// TwinCAT 3 PLC project Perlage_Standard
// libraries:
//   Recipe Management, * (System)
//   Tc2_Drive, * (Beckhoff Automation GmbH)
//   Tc2_EtherCAT, * (Beckhoff Automation GmbH)
//   Tc2_Math, * (Beckhoff Automation GmbH)
//   Tc2_MC2, * (Beckhoff Automation GmbH)
//   Tc2_MC2_Drive, * (Beckhoff Automation GmbH)
//   Tc2_NC, * (Beckhoff Automation GmbH)
//   Tc2_SerialCom, * (Beckhoff Automation GmbH)
//   Tc2_Standard, * (Beckhoff Automation GmbH)
//   Tc2_Standard, * (Beckhoff Automation GmbH)
//   Tc2_System, * (Beckhoff Automation GmbH)
//   Tc2_System, * (Beckhoff Automation GmbH)
//   Tc2_Utilities, * (Beckhoff Automation GmbH)
//   Tc3_Module, * (Beckhoff Automation GmbH)
//   Tc3_Module, * (Beckhoff Automation GmbH)
// project tree:
//   Data types/ TAutoSampling.TcDUT, TAxisCommands.TcDUT, TAxisHomingType.TcDUT, TAxisState.TcDUT, TAxisType.TcDUT, TComIndex.TcDUT, TConfigFileData.TcDUT, TCounter.TcDUT, TDashboardCmd.TcDUT, TDataLog.TcDUT, TDynAxisParam.TcDUT, TErrors.TcDUT, TGiver.TcDUT, THolderIndex.TcDUT, TLiftPos.TcDUT, TLiftType.TcDUT, TLoaderAxis.TcDUT, TLoaderDropMode.TcDUT, TLoaderHead.TcDUT, TLoaderModulePos.TcDUT, TLoaderPlatePos.TcDUT, TLoaderSynchro.TcDUT, TLoaderTakeMode.TcDUT, TLoaderTeachedAxis.TcDUT, TLoaderTeachOffset.TcDUT, TLoaderTeachPos.TcDUT, TMachineData.TcDUT, TMachineManual.TcDUT, TMachineMode.TcDUT, TMachineModeMask.TcDUT, TMachineOptions.TcDUT, TMachineSafety.TcDUT, TManagerPartStatus.TcDUT, TManBarrel.TcDUT, TManBarrelAxisPosition.TcDUT, TManButton.TcDUT, TManDrive.TcDUT, TManDrivePos.TcDUT, TManLift.TcDUT, TManLoader.TcDUT, TManPearling.TcDUT, TManReject.TcDUT, TManSharpen.TcDUT, TManTable.TcDUT, TManTurnOver.TcDUT, TManualData.TcDUT, TManUtilities.TcDUT, TManVision.TcDUT, TMCRCommands.TcDUT, TMDE.TcDUT, TMDEStatus.TcDUT, TMMIPearlData.TcDUT, TModuleCommands.TcDUT, TModuleData.TcDUT, TModuleStatus.TcDUT, TModuleSteps.TcDUT, TOperatorReq.TcDUT, TPartData.TcDUT, TPartDataMMI.TcDUT, TPearlingAxis.TcDUT, TPearlingData.TcDUT, TPearlingDataHead.TcDUT, TPearlingDebug.TcDUT, TPearlingHead.TcDUT, TPearlingSide.TcDUT, TPearlingTeachPos.TcDUT, TPearlsArea.TcDUT, TPearlsTable.TcDUT, TPlateData.TcDUT, TPlatePartStatus.TcDUT, TPositionXY.TcDUT, TPositionXYTheta.TcDUT, TProbingArea.TcDUT, TProbingLog.TcDUT, TprodCounter.TcDUT, TProductionCmd.TcDUT, TProductionLot.TcDUT, TProductionStats.TcDUT, TRejectReason.TcDUT (excluded from build), TRejectStatus.TcDUT, TRobotPos.TcDUT, TRunCmdBarrel.TcDUT, TRunCmdLift.TcDUT, TRunCmdLoader.TcDUT, TRunCmdPearling.TcDUT, TRunCmdReject.TcDUT, TRunCmdSharpen.TcDUT, TRunCmdTable.TcDUT, TRunCmdTurnOver.TcDUT, TRunCmdVision.TcDUT, TRunData.TcDUT, TRunDataLift.TcDUT, TRunDataLoader.TcDUT, TRunDataPearling.TcDUT, TRunDataPlate.TcDUT, TRunDataReject.TcDUT, TRunDataTable.TcDUT, TRunDataTurnOver.TcDUT, TRunDataVision.TcDUT, TRunStatus.TcDUT, TStationGiversTakers.TcDUT, TStationIndex.TcDUT, TStickData.TcDUT, TStickDataMMI.TcDUT, TStickDataMMIShared.TcDUT, TStickDataShared.TcDUT, TTableSide.TcDUT, TTaker.TcDUT, TTransferIndex.TcDUT, TTurnOverPos.TcDUT, TVaccumSettings.TcDUT, TVacuumSettingsMMI.TcDUT, TVisionData.TcDUT, TVisionPartData.TcDUT, TVisionRequest.TcDUT
//   / FastTaskForRS.TcTTO, Recipe Manager.TcRMO (not stored), Standard.TcTTO
//   Global Variables/ Global_Variables.TcGVL, TwinCAT_Configuration.TcGVL, Variable_Configuration.TcGVL
//   POUs/ BG_Serial.TcPOU, MAIN.TcPOU
//   POUs/Controls/ FB_AspirationValve.TcPOU, FB_CheckJack1_1.TcPOU, FB_CheckJack1_2.TcPOU, FB_CheckJack2_2.TcPOU, FB_Vacuum.TcPOU, FB_VacuumAnalogCheck.TcPOU
//   POUs/Drivers/ MCRDrv.TcPOU, StdAxis.TcPOU
//   POUs/Handlers/ BarrelHdl.TcPOU, LiftHdl.TcPOU, LoaderHdl.TcPOU, PearlingHdl.TcPOU, RejectHdl.TcPOU, SharpenHdl.TcPOU, TableHdl.TcPOU, TurnOverHdl.TcPOU, UtilitiesHdl.TcPOU, VisionHdl.TcPOU
//   POUs/Manager/ Manager.TcPOU, ManagerDashboard.TcPOU, ManagerRun.TcPOU, ManagerRunTest.TcPOU
//   POUs/utils/ CalculatePosAngle.TcPOU, ComputeVisionPos.TcPOU, ConverterLinearLimit.TcPOU, Dispersion.TcPOU, GetLoaderAxisFromTeachedAxis.TcPOU, GetLoaderTeachedAxisFromAxis.TcPOU, HandleErrors.TcPOU, yGetActiveSection.TcPOU, InitNewPartData.TcPOU, MTBFCounter.TcPOU, RunningCounter.TcPOU, StopWatch.TcPOU, TBlink.TcPOU, yCalcCheckSum.TcPOU
// real-time tasks:
//   TASK FastTaskForRS: cycle T#2ms, priority 21, ADS port 350
//   TASK Standard: cycle T#4ms, priority 20, ADS port 351
// motion (NC):
//   TASK NC-Task 1 SAF: cycle T#2ms, priority 4, ADS port 501
//   TASK NC-Task 1 SVB: cycle T#10ms, priority 8, ADS port 511
//   AXIS Loader X (id 42)
//     Dynamic: AccelerationMaximum=0, DecelerationMaximum=0, Acceleration=12400, Deceleration=12400, Jerk=248000, DelayTime=0.004
//     Velo: RefSearch=50, RefSync=14.65, SlowManual=15, FastManual=50, Fast=1465.10989583333, Maximum=620
//     TargetPosControl: Range=0.01
//     encoder EncType=8
//       EncPara: ScaleFactorNumerator=16, ScaleFactorDenominator=1048576, Inverse=true, MaxCount=#xffffffff
//         SoftEndMinControl: Enable=true, Range=-20
//         SoftEndMaxControl: Enable=true, Range=680
//         Inc: RefSearchInverse=true, RefSyncInverse=false, RefMode=5
//     drive DrvType=9
//       DrvPara: Inverse=true, MaxCount=#xffffffff, DriveControlDWord=#x00030100
//         Analog: VeloReferenz=1611.62088541667, VeloScale=1.02400649589962, SmoothingFilterOrder=0, SmoothingFilterTime=0
//         TimeComp: TaskDelayCycles=1
//     controller CtrType=1
//       CtrPara: PriorControlFactor=1
//         PosDiffControl: Range=1
//         PID: PosKp=10
//         Observer: BandWidth=20
//   AXIS Loader Y (id 43)
//     Dynamic: AccelerationMaximum=0, DecelerationMaximum=0, Acceleration=12400, Deceleration=12400, Jerk=248000, DelayTime=0.004
//     Velo: RefSearch=50, RefSync=14.65, SlowManual=15, FastManual=50, Fast=1465.10989583333, Maximum=620
//     TargetPosControl: Range=0.01
//     encoder EncType=8
//       EncPara: ScaleFactorNumerator=16, ScaleFactorDenominator=1048576, MaxCount=#xffffffff
//         SoftEndMinControl: Enable=true, Range=-14
//         SoftEndMaxControl: Enable=true, Range=475
//         Inc: RefSearchInverse=true, RefSyncInverse=false, RefMode=5
//     drive DrvType=9
//       DrvPara: MaxCount=#xffffffff, DriveControlDWord=#x00030100
//         Analog: VeloReferenz=1611.62088541667, VeloScale=1.02400649589962, SmoothingFilterOrder=0, SmoothingFilterTime=0
//         TimeComp: TaskDelayCycles=1
//     controller CtrType=1
//       CtrPara: PriorControlFactor=1
//         PosDiffControl: Range=1
//         PID: PosKp=10
//         Observer: BandWidth=20
//   AXIS Loader Z1 (id 5)
//     Dynamic: AccelerationMaximum=1500, DecelerationMaximum=1500, Acceleration=215, Deceleration=215, Jerk=153752
//     Velo: RefSearch=3, RefSync=3, SlowManual=10, FastManual=10, Fast=300, Maximum=35
//     TargetPosControl: Range=0.1
//     OtherSettings: AllowMotionCmdToSlave=true
//     encoder EncType=19
//       EncPara: ScaleFactorNumerator=3, ScaleFactorDenominator=1048576, MaxCount=#xffffffff
//         SoftEndMinControl: Enable=true, Range=-12
//         SoftEndMaxControl: Enable=true, Range=13.5
//         Inc: RefSearchInverse=true, RefSyncInverse=false, RefMode=5
//     drive DrvType=16
//       DrvPara: MaxCount=#xffffffff, DriveControlDWord=#x00020000
//         Analog: VeloReferenz=330, VeloScale=32, ScaleFactorActTorque=0.1
//         TimeComp: TaskDelayCycles=1
//     controller CtrType=1
//       CtrPara: PriorControlFactor=1
//         PID: PosKp=10
//         Observer: BandWidth=20
//   AXIS Loader Z2 (id 6)
//     Dynamic: AccelerationMaximum=1500, DecelerationMaximum=1500, Acceleration=215, Deceleration=215, Jerk=153752
//     Velo: RefSearch=3, RefSync=3, SlowManual=10, FastManual=10, Fast=300, Maximum=35
//     TargetPosControl: Range=0.1
//     OtherSettings: AllowMotionCmdToSlave=true
//     encoder EncType=19
//       EncPara: ScaleFactorNumerator=3, ScaleFactorDenominator=1048576, MaxCount=#xffffffff
//         SoftEndMinControl: Enable=true, Range=-12.8
//         SoftEndMaxControl: Enable=true, Range=13
//         Inc: RefSearchInverse=true, RefSyncInverse=false, RefMode=5
//     drive DrvType=16
//       DrvPara: MaxCount=#xffffffff, DriveControlDWord=#x00020000
//         Analog: VeloReferenz=330, VeloScale=32, ScaleFactorActTorque=0.1
//         TimeComp: TaskDelayCycles=1
//     controller CtrType=1
//       CtrPara: PriorControlFactor=1
//         PID: PosKp=10
//         Observer: BandWidth=20
//   AXIS Loader Theta (id 8)
//     General: UnitName=°, UnitFlags=#x00000004
//     Dynamic: AccelerationMaximum=0, DecelerationMaximum=0, Acceleration=72000, Deceleration=72000, Jerk=1440000, DelayTime=0.004
//     Velo: RefSearch=1, RefSync=200, SlowManual=50, FastManual=200, Maximum=400
//     TargetPosControl: Range=0.1
//     encoder EncType=4
//       EncPara: ScaleFactorNumerator=0.0439453125, MaxCount=#x00001fff
//         Inc: RefSyncInverse=false, RefSoftSyncMask=#x00001fff
//     drive DrvType=24
//       DrvPara: Inverse=true
//         Analog: VeloReferenz=3600, SmoothingFilterOrder=0, SmoothingFilterTime=0
//         TimeComp: TaskDelayCycles=1
//     controller CtrType=2
//       CtrPara: PriorControlFactor=1
//         PID: PosKp=15
//         Observer: BandWidth=20
//   AXIS Lift1 (id 4)
//     Dynamic: AccelerationMaximum=0, DecelerationMaximum=0, Acceleration=400, Deceleration=400, Jerk=4000, DelayTime=0.004
//     Velo: RefSearch=10, RefSync=1, SlowManual=10, FastManual=20, Fast=156.08333333231, Maximum=40
//     PositionAreaControl: Range=0.2
//     TargetPosControl: Range=0.1
//     encoder EncType=19
//       EncPara: ScaleFactorNumerator=1.66666666665574, ScaleFactorDenominator=1048576, MaxCount=#xffffffff
//         SoftEndMinControl: Enable=true, Range=-33
//         SoftEndMaxControl: Enable=true, Range=240
//         Inc: RefSearchInverse=true, RefSyncInverse=false, RefMode=5
//     drive DrvType=16
//       DrvPara: MaxCount=#xffffffff, DriveControlDWord=#x00020000
//         Analog: VeloReferenz=171.691666665541, VeloScale=32, SmoothingFilterOrder=0, SmoothingFilterTime=0
//         TimeComp: TaskDelayCycles=1
//     controller CtrType=1
//       CtrPara: PriorControlFactor=1
//         PosDiffControl: Range=1
//         PID: PosKp=10
//         Observer: BandWidth=20
//   AXIS Lift2 (id 1)
//     Dynamic: AccelerationMaximum=0, DecelerationMaximum=0, Acceleration=400, Deceleration=400, Jerk=4000, DelayTime=0.004
//     Velo: RefSearch=10, RefSync=1, SlowManual=10, FastManual=20, Fast=145.027777776827, Maximum=40
//     PositionAreaControl: Range=0.2
//     TargetPosControl: Range=0.1
//     encoder EncType=19
//       EncPara: ScaleFactorNumerator=1.66666666665574, ScaleFactorDenominator=1048576, MaxCount=#xffffffff
//         SoftEndMinControl: Enable=true, Range=-33
//         SoftEndMaxControl: Enable=true, Range=240
//         Inc: RefSearchInverse=true, RefSyncInverse=false, RefMode=5
//     drive DrvType=16
//       DrvPara: MaxCount=#xffffffff, DriveControlDWord=#x00020000
//         Analog: VeloReferenz=159.53055555451, VeloScale=32, SmoothingFilterOrder=0, SmoothingFilterTime=0
//         TimeComp: TaskDelayCycles=1
//     controller CtrType=1
//       CtrPara: PriorControlFactor=1
//         PosDiffControl: Range=1
//         PID: PosKp=10
//         Observer: BandWidth=20
//   AXIS Table (id 13)
//     General: UnitName=°
//     Dynamic: AccelerationMaximum=0, DecelerationMaximum=0, Acceleration=10000, Deceleration=10000, Jerk=10000, DelayTime=0.004
//     Velo: RefSearch=10, RefSync=5, SlowManual=20, FastManual=50, Fast=1645.2, Maximum=360
//     PositionAreaControl: Range=0.5
//     TargetPosControl: Range=0.5, Time=0.1
//     encoder EncType=8
//       EncPara: ScaleFactorNumerator=3.4332275391e-05, MaxCount=#xffffffff
//         SoftEndMinControl: Enable=true, Range=-28
//         SoftEndMaxControl: Enable=true, Range=155
//         Inc: RefSearchInverse=true, RefSyncInverse=false, RefMode=5
//     drive DrvType=9
//       DrvPara: MaxCount=#xffffffff, DriveControlDWord=#x00030100
//         Analog: VeloReferenz=1809.72, VeloScale=1.02400649589962, SmoothingFilterOrder=0, SmoothingFilterTime=0
//         TimeComp: TaskDelayCycles=1
//     controller CtrType=1
//       CtrPara: PriorControlFactor=1
//         PosDiffControl: Range=1
//         PID: PosKp=10
//         Observer: BandWidth=20
//   AXIS Pearling X (id 40)
//     Dynamic: AccelerationMaximum=0, DecelerationMaximum=0, Jerk=22500, DelayTime=0.004
//     Velo: RefSearch=20, RefSync=4.57846842447917, SlowManual=10, FastManual=10, Fast=457.846842447917, Maximum=200
//     TargetPosControl: Range=0.015
//     encoder EncType=8
//       EncPara: ScaleFactorNumerator=5, ScaleFactorDenominator=1048576, Inverse=true, MaxCount=#xffffffff
//         SoftEndMinControl: Enable=true, Range=-19
//         SoftEndMaxControl: Enable=true, Range=380
//         Inc: RefSearchInverse=true, RefSyncInverse=false, RefMode=5
//     drive DrvType=9
//       DrvPara: Inverse=true, MaxCount=#xffffffff, DriveControlDWord=#x00030100
//         Analog: VeloReferenz=503.631526692708, VeloScale=1.02400649589962, SmoothingFilterOrder=0, SmoothingFilterTime=0
//         TimeComp: TaskDelayCycles=1
//     controller CtrType=1
//       CtrPara: PriorControlFactor=1
//         Observer: BandWidth=20
//   AXIS Pearling Y (id 41)
//     Dynamic: AccelerationMaximum=0, DecelerationMaximum=0, Jerk=22500, DelayTime=0.004
//     Velo: RefSearch=20, RefSync=4.57846842447917, SlowManual=10, FastManual=10, Fast=457.846842447917, Maximum=200
//     TargetPosControl: Range=0.015
//     encoder EncType=8
//       EncPara: ScaleFactorNumerator=5, ScaleFactorDenominator=1048576, Inverse=true, MaxCount=#xffffffff
//         SoftEndMinControl: Enable=true, Range=-16
//         SoftEndMaxControl: Enable=true, Range=90
//         Inc: RefSearchInverse=true, RefSyncInverse=false, RefMode=5
//     drive DrvType=9
//       DrvPara: Inverse=true, MaxCount=#xffffffff, DriveControlDWord=#x00030100
//         Analog: VeloReferenz=503.631526692708, VeloScale=1.02400649589962, SmoothingFilterOrder=0, SmoothingFilterTime=0
//         TimeComp: TaskDelayCycles=1
//     controller CtrType=1
//       CtrPara: PriorControlFactor=1
//         Observer: BandWidth=20
//   AXIS Pearling Z1 (id 12)
//     Dynamic: Acceleration=3200, Deceleration=3200, Jerk=170667
//     Velo: RefSearch=20, RefSync=5, SlowManual=5.8, FastManual=12, Fast=116, Maximum=100
//     OtherSettings: AllowMotionCmdToSlave=true
//     encoder EncType=19
//       EncPara: ScaleFactorNumerator=2, ScaleFactorDenominator=1048576, MaxCount=#xffffffff
//         SoftEndMinControl: Enable=true, Range=-19
//         SoftEndMaxControl: Enable=true, Range=55
//         Inc: RefSearchInverse=true, RefSyncInverse=false, RefMode=5
//     drive DrvType=16
//       DrvPara: MaxCount=#xffffffff, DriveControlDWord=#x00020000
//         Analog: VeloReferenz=127.6, VeloScale=32, ScaleFactorActTorque=0.1
//         TimeComp: TaskDelayCycles=1
//     controller CtrType=1
//       CtrPara: PriorControlFactor=1
//         PID: PosKp=10
//         Observer: BandWidth=20
//   AXIS Pearling Z2 (id 14)
//     Dynamic: Acceleration=3200, Deceleration=3200, Jerk=170667
//     Velo: RefSearch=20, RefSync=5, SlowManual=5.8, FastManual=12, Fast=116, Maximum=100
//     OtherSettings: AllowMotionCmdToSlave=true
//     encoder EncType=19
//       EncPara: ScaleFactorNumerator=2, ScaleFactorDenominator=1048576, MaxCount=#xffffffff
//         SoftEndMinControl: Enable=true, Range=-19
//         SoftEndMaxControl: Enable=true, Range=55
//         Inc: RefSearchInverse=true, RefSyncInverse=false, RefMode=5
//     drive DrvType=16
//       DrvPara: MaxCount=#xffffffff, DriveControlDWord=#x00020000
//         Analog: VeloReferenz=127.6, VeloScale=32, ScaleFactorActTorque=0.1
//         TimeComp: TaskDelayCycles=1
//     controller CtrType=1
//       CtrPara: PriorControlFactor=1
//         PID: PosKp=10
//         Observer: BandWidth=20
//   AXIS Barrel (id 10)
//     General: UnitName=°, UnitFlags=#x00000004
//     Dynamic: AccelerationMaximum=0, DecelerationMaximum=0, Acceleration=300, Deceleration=300, Jerk=500000, DelayTime=0.004
//     Velo: RefSearch=15, RefSync=200, FastManual=200, Maximum=200
//     TargetPosControl: Range=0.5
//     encoder EncType=4
//       EncPara: ScaleFactorNumerator=0.087890625, Inverse=true, MaxCount=#x00000fff
//         Inc: RefMode=2, RefSoftSyncMask=#x000003ff
//     drive DrvType=24
//       DrvPara: Inverse=true
//         Analog: VeloReferenz=3600, SmoothingFilterOrder=0, SmoothingFilterTime=0
//         TimeComp: TaskDelayCycles=1
//     controller CtrType=1
//       CtrPara: PriorControlFactor=1
//         PID: VeloKp=0
//         Observer: BandWidth=20
//   AXIS Sharpen (id 9)
//     Dynamic: AccelerationMaximum=0, DecelerationMaximum=0, Acceleration=22.1997, Deceleration=22.1997, Jerk=985.643, DelayTime=0.004
//     Velo: SlowManual=10, FastManual=10, Maximum=10
//     encoder EncType=1
//       EncPara: ScaleFactorNumerator=62.8, ScaleFactorDenominator=4096
//         Inc: RefSoftSyncMask=#x0000ffff
//     drive DrvType=24
//       Analog: VeloReferenz=363.5271499, SmoothingFilterOrder=0, SmoothingFilterTime=0
//       TimeComp: TaskDelayCycles=1
//     controller CtrType=1
//       CtrPara: PriorControlFactor=1
//         PosDiffControl: Range=10
//         Observer: BandWidth=20
//   AXIS SharpenEncoder (id 3)
//     Dynamic: AccelerationMaximum=0, DecelerationMaximum=0
//     encoder EncType=4
//       EncPara: ScaleFactorNumerator=62.8, ScaleFactorDenominator=1024, MaxCount=#x0000ffff
//         Inc: RefMode=2, RefSoftSyncMask=#x0000ffff
//     drive DrvType=5
//       Analog: SmoothingFilterOrder=0, SmoothingFilterTime=0
//       TimeComp: TaskDelayCycles=1
//     controller CtrType=1
//       CtrPara: PriorControlFactor=1
//         Observer: BandWidth=20
//   AXIS Brush (id 7)
//     General: UnitName=°
//     Dynamic: AccelerationMaximum=0, DecelerationMaximum=0, Acceleration=4710, Deceleration=4710, Jerk=12973.2, DelayTime=0.004
//     Velo: RefSearch=31.3285714286399, RefSync=31.3285714286399, SlowManual=156.642857143199, FastManual=939.857142859196, Fast=3132.85714286399, Maximum=3000
//     TargetPosControl: Range=0.5
//     encoder EncType=19
//       EncPara: ScaleFactorNumerator=85.714285714473, ScaleFactorDenominator=1048576, MaxCount=#xffffffff
//         SoftEndMinControl: Enable=true, Range=-108
//         SoftEndMaxControl: Enable=true, Range=50
//         Inc: RefSearchInverse=true, RefSyncInverse=false, RefMode=5
//     drive DrvType=16
//       DrvPara: MaxCount=#xffffffff
//         Analog: VeloReferenz=3446.14285715039, VeloScale=32, SmoothingFilterOrder=0, SmoothingFilterTime=0
//         TimeComp: TaskDelayCycles=1
//     controller CtrType=3
//       CtrPara: PriorControlFactor=1
//         PID: PosKp=5
//         Observer: BandWidth=20
// I/O:
//   DEVICE Device 2 (EtherCAT) (disabled), AmsNetId 172.16.1.155.3.1
//     A18.1 (PeAxMotor PeAyMotor) [AX5203-0000-0203 EtherCAT Drive (SoE, 2 Ch.)]
//     A18.2 (PoAxMotor PoAyMotor) [AX5203-0000-0203 EtherCAT Drive (SoE, 2 Ch.)]
//     A18.3 Table (AX5203-0000-0203) [AX5203-0000-0203 EtherCAT Drive (SoE, 2 Ch.)]
//     A22.A (Term IO) [EK1100 EtherCAT Coupler (2A E-Bus)]
//       A22.1 [EL1809 16Ch. Dig. Input 24V, 3ms]
//       A22.2 [EL1809 16Ch. Dig. Input 24V, 3ms]
//       A22.3 [EL1809 16Ch. Dig. Input 24V, 3ms]
//       A22.4 [EL1809 16Ch. Dig. Input 24V, 3ms]
//       A23.1 [EL1008 8Ch. Dig. Input 24V, 3ms]
//       A25.1 [EL3044 4Ch. Ana. Input 0-20mA]
//       A25.2 [EL3044 4Ch. Ana. Input 0-20mA]
//       A25.4 [EL3044 4Ch. Ana. Input 0-20mA]
//       A25.A [EL9505 Power supply terminal 5V]
//       A25.3 [EL3062 2Ch. Ana. Input 0-10V]
//       A26.A [EL9100 Power Supplier with LED (24V)]
//       A26.1 [EL2024 4Ch. Dig. Output 24V, 2A]
//       A26.2 [EL2809 16Ch. Dig. Output 24V, 0.5A]
//       A28.A [EL9100 Power Supplier with LED (24V)]
//       A28.1 [EL2004 4Ch. Dig. Output 24V, 0.5A]
//       A29.A [EL9410 E-Bus Power Supplier  (Diagnostics)]
//       A29.1 (Twinsafe PLC) [EL1918, 8Ch. Safety Input 24V, TwinSAFE]
//         modules: Module 2 (FSLOGIC)
//       A29.4 (TwinSafe IN) [EL1904, 4 Ch. Safety Input 24V, TwinSAFE]
//         modules: Module 1 (FSOES)
//       A29.5 (TwinSafe OUT) [EL2904, 4 Ch. Safety Output 24V, 0.5A, TwinSAFE]
//         modules: Module 1 (FSOES), Module 2 (DO)
//       A31.B [EL9576 Brake chopper terminal]
//       A31.1 (Lf1CmdMotor)_old [EL7201-0010 1Ch. MDP742 Servo motor output stage with OCT (50V, 4A)] (disabled)
//       A31.1 (Lf1CmdMotor) [EL7201-0010 1Ch. MDP742 Servo motor output stage with OCT (50V, 2.8A RMS)]
//       A31.2 (Lf2CmdMotor)_old [EL7201-0010 1Ch. MDP742 Servo motor output stage with OCT (50V, 2.8A RMS)] (disabled)
//       A31.2 (Lf2CmdMotor) [EL7201-0010 1Ch. MDP742 Servo motor output stage with OCT (50V, 2.8A RMS)]
//       A31.C [EL9576 Brake chopper terminal]
//       A31.3 (PeZ1CmdMotor) [EL7211 1Ch. MDP742 Servo motor output stage (50V, 4.5A RMS)]
//       A31.4 (PeZ2CmdMotor) [EL7211 1Ch. MDP742 Servo motor output stage (50V, 4.5A RMS)]
//       A32.A [EL9576 Brake chopper terminal]
//       A32.1 (PeBrCmdMotor) [EL7211 1Ch. MDP742 Servo motor output stage (50V, 4.5A RMS)]
//       A33.A [EL9576 Brake chopper terminal]
//       A33.1 (PoAz1MotCmd) [EL7201 1Ch. MDP742 Servo motor output stage (50V, 4A)]
//       A33.2 (PoAz2MotCmd) [EL7201 1Ch. MDP742 Servo motor output stage (50V, 4A)]
//       A33.C [EL9410 E-Bus Power Supplier  (Diagnostics)]
//       A33.B [EL9576 Brake chopper terminal]
//       A33.3 (PoAtCmdMotor) [EL7047 1Ch. Stepper motor output stage (50V, 5A)]
//       A33.4 (ReCmdMotor) [EL7047 1Ch. Stepper motor output stage (50V, 5A)]
//       A34.A [EL9576 Brake chopper terminal]
//       A34.1 (ShCmdMotor) [EL7047 1Ch. Stepper motor output stage (50V, 5A)]
//       A34.2 (BaCmdMotor) [EL7047 1Ch. Stepper motor output stage (50V, 5A)]
//       A34.E [EL9011 End Terminal]
//     A75.1 [EX260-SEC1 EtherCAT SI Unit (32DO_PNP) Rev1.2]
//     A79.1 [EX260-SEC1 EtherCAT SI Unit (32DO_PNP) Rev1.2]
//     A79.2 [EX260-SEC1 EtherCAT SI Unit (32DO_PNP) Rev1.2]
// variable links:
//   Device 2 (EtherCAT) <-> Device 2 (EtherCAT)/A22.A (Term IO)/A29.1 (Twinsafe PLC)
//     A22.A (Term IO)/A29.4 (TwinSafe IN)/Module 1 (FSOES)/RxPDO/FSOE <-> ConnectionInputs/TwinSafeGroup1.A29_4_2 TxPDO
//   Device 2 (EtherCAT) <-> Device 2 (EtherCAT)/A22.A (Term IO)/A29.4 (TwinSafe IN)
//     A22.A (Term IO)/A29.1 (Twinsafe PLC)/ConnectionOutputs/TwinSafeGroup1.A29_4_2 RxPDO <-> Module 1 (FSOES)/TxPDO/FSOE
//   Device 2 (EtherCAT) <-> Device 2 (EtherCAT)/A22.A (Term IO)/A29.5 (TwinSafe OUT)
//     A22.A (Term IO)/A29.1 (Twinsafe PLC)/ConnectionInputs/TwinSafeGroup1.A29_5_3 TxPDO <-> Module 1 (FSOES)/RxPDO/FSOE
//     A22.A (Term IO)/A29.1 (Twinsafe PLC)/ConnectionOutputs/TwinSafeGroup1.A29_5_3 RxPDO <-> Module 1 (FSOES)/TxPDO/FSOE
//   NC-Task 1 SAF/Axes/Barrel <-> Device 2 (EtherCAT)/A22.A (Term IO)/A34.2 (BaCmdMotor)
//     Barrel_Drive/Inputs/Barrel_Drive_In/nState1 @bit 3 <-> STM Status/Status/Error
//     Barrel_Drive/Inputs/Barrel_Drive_In/nState1 @bit 7 <-> STM Status/Status/Motor stall
//     Barrel_Drive/Inputs/Barrel_Drive_In/nState1 @bit 5 <-> STM Status/Status/Moving negative
//     Barrel_Drive/Inputs/Barrel_Drive_In/nState1 @bit 4 <-> STM Status/Status/Moving positive
//     Barrel_Drive/Inputs/Barrel_Drive_In/nState1 @bit 1 <-> STM Status/Status/Ready
//     Barrel_Drive/Inputs/Barrel_Drive_In/nState1 <-> STM Status/Status/Ready to enable
//     Barrel_Drive/Inputs/Barrel_Drive_In/nState1 @bit 6 <-> STM Status/Status/Torque reduced
//     Barrel_Drive/Inputs/Barrel_Drive_In/nState1 @bit 2 <-> STM Status/Status/Warning
//     Barrel_Drive/Inputs/Barrel_Drive_In/nState2 @bit 3 <-> STM Status/Status/Digital input 1
//     Barrel_Drive/Inputs/Barrel_Drive_In/nState2 @bit 4 <-> STM Status/Status/Digital input 2
//     Barrel_Drive/Inputs/Barrel_Drive_In/nState2 @bit 5 <-> STM Status/Status/Sync error
//     Barrel_Drive/Inputs/Barrel_Drive_In/nState2 @bit 7 <-> STM Status/Status/TxPDO Toggle
//     Barrel_Drive/Inputs/Barrel_Drive_In/nState4 @bit 1 <-> WcState/InputToggle
//     Barrel_Drive/Inputs/Barrel_Drive_In/nState4 <-> WcState/WcState
//     Barrel_Drive/Outputs/Barrel_Drive_Out/nCtrl1 <-> STM Control/Control/Enable
//     Barrel_Drive/Outputs/Barrel_Drive_Out/nCtrl1 @bit 2 <-> STM Control/Control/Reduce torque
//     Barrel_Drive/Outputs/Barrel_Drive_Out/nCtrl1 @bit 1 <-> STM Control/Control/Reset
//     Barrel_Drive/Outputs/Barrel_Drive_Out/nCtrl2 @bit 3 <-> STM Control/Control/Digital output 1
//     Barrel_Drive/Outputs/Barrel_Drive_Out/nDataOut2[0] <-> STM Velocity/Velocity
//     Barrel_Enc/Inputs/Barrel_Enc_In/nDataIn1[0] <-> ENC Status compact/Counter value
//     Barrel_Enc/Inputs/Barrel_Enc_In/nDataIn2[0] <-> ENC Status compact/Latch value
//     Barrel_Enc/Inputs/Barrel_Enc_In/nState1 @bit 4 <-> ENC Status compact/Status/Counter overflow
//     Barrel_Enc/Inputs/Barrel_Enc_In/nState1 @bit 3 <-> ENC Status compact/Status/Counter underflow
//     Barrel_Enc/Inputs/Barrel_Enc_In/nState1 @bit 7 <-> ENC Status compact/Status/Extrapolation stall
//     Barrel_Enc/Inputs/Barrel_Enc_In/nState1 <-> ENC Status compact/Status/Latch C valid
//     Barrel_Enc/Inputs/Barrel_Enc_In/nState1 @bit 1 <-> ENC Status compact/Status/Latch extern valid
//     Barrel_Enc/Inputs/Barrel_Enc_In/nState1 @bit 2 <-> ENC Status compact/Status/Set counter done
//     Barrel_Enc/Inputs/Barrel_Enc_In/nState2 @bit 4 <-> ENC Status compact/Status/Status of extern latch
//     Barrel_Enc/Inputs/Barrel_Enc_In/nState2 <-> ENC Status compact/Status/Status of input A
//     Barrel_Enc/Inputs/Barrel_Enc_In/nState2 @bit 1 <-> ENC Status compact/Status/Status of input B
//     Barrel_Enc/Inputs/Barrel_Enc_In/nState2 @bit 2 <-> ENC Status compact/Status/Status of input C
//     Barrel_Enc/Inputs/Barrel_Enc_In/nState2 @bit 5 <-> ENC Status compact/Status/Sync error
//     Barrel_Enc/Inputs/Barrel_Enc_In/nState2 @bit 7 <-> ENC Status compact/Status/TxPDO Toggle
//     Barrel_Enc/Inputs/Barrel_Enc_In/nState4 @bit 1 <-> WcState/InputToggle
//     Barrel_Enc/Inputs/Barrel_Enc_In/nState4 <-> WcState/WcState
//     Barrel_Enc/Outputs/Barrel_Enc_Out/nCtrl1 <-> ENC Control compact/Control/Enable latch C
//     Barrel_Enc/Outputs/Barrel_Enc_Out/nCtrl1 @bit 3 <-> ENC Control compact/Control/Enable latch extern on negative edge
//     Barrel_Enc/Outputs/Barrel_Enc_Out/nCtrl1 @bit 1 <-> ENC Control compact/Control/Enable latch extern on positive edge
//     Barrel_Enc/Outputs/Barrel_Enc_Out/nCtrl1 @bit 2 <-> ENC Control compact/Control/Set counter
//     Barrel_Enc/Outputs/Barrel_Enc_Out/nDataOut1[0] <-> ENC Control compact/Set counter value
//   NC-Task 1 SAF/Axes/Brush <-> Device 2 (EtherCAT)/A22.A (Term IO)/A32.1 (PeBrCmdMotor)
//     Brush_Drive/Inputs/Brush_Drive_In/nDcOutputTime <-> InfoData/DcOutputShift
//     Brush_Drive/Inputs/Brush_Drive_In/nState1 <-> DRV Statusword/Statusword
//     Brush_Drive/Inputs/Brush_Drive_In/nState2 <-> DRV Statusword/Statusword @bit 8
//     Brush_Drive/Inputs/Brush_Drive_In/nState4 @bit 1 <-> WcState/InputToggle
//     Brush_Drive/Inputs/Brush_Drive_In/nState4 <-> WcState/WcState
//     Brush_Drive/Outputs/Brush_Drive_Out/nCtrl1 <-> DRV Controlword/Controlword
//     Brush_Drive/Outputs/Brush_Drive_Out/nCtrl2 <-> DRV Controlword/Controlword @bit 8
//     Brush_Drive/Outputs/Brush_Drive_Out/nDataOut2 <-> DRV Target velocity/Target velocity
//     Brush_Enc/Inputs/Brush_Enc_In/nDataIn1 <-> FB Position/Position
//     Brush_Enc/Inputs/Brush_Enc_In/nDcInputTime <-> InfoData/DcInputShift
//     Brush_Enc/Inputs/Brush_Enc_In/nState4 @bit 1 <-> WcState/InputToggle
//     Brush_Enc/Inputs/Brush_Enc_In/nState4 <-> WcState/WcState
//   NC-Task 1 SAF/Axes/Lift1 <-> Device 2 (EtherCAT)/A22.A (Term IO)/A31.1 (Lf1CmdMotor)
//     Lift1_Drive/Inputs/Lift1_Drive_In/nDcOutputTime <-> InfoData/DcOutputShift
//     Lift1_Drive/Inputs/Lift1_Drive_In/nState1 <-> DRV Statusword/Statusword
//     Lift1_Drive/Inputs/Lift1_Drive_In/nState2 <-> DRV Statusword/Statusword @bit 8
//     Lift1_Drive/Inputs/Lift1_Drive_In/nState4 @bit 1 <-> WcState/InputToggle
//     Lift1_Drive/Inputs/Lift1_Drive_In/nState4 <-> WcState/WcState
//     Lift1_Drive/Outputs/Lift1_Drive_Out/nCtrl1 <-> DRV Controlword/Controlword
//     Lift1_Drive/Outputs/Lift1_Drive_Out/nCtrl2 <-> DRV Controlword/Controlword @bit 8
//     Lift1_Drive/Outputs/Lift1_Drive_Out/nDataOut2 <-> DRV Target velocity/Target velocity
//     Lift1_Enc/Inputs/Lift1_Enc_In/nDataIn1 <-> FB Position/Position
//     Lift1_Enc/Inputs/Lift1_Enc_In/nDcInputTime <-> InfoData/DcInputShift
//     Lift1_Enc/Inputs/Lift1_Enc_In/nState4 @bit 1 <-> WcState/InputToggle
//     Lift1_Enc/Inputs/Lift1_Enc_In/nState4 <-> WcState/WcState
//     Lift1_Enc/Inputs/Lift1_Enc_In/nState5 <-> FB Touch probe status/Touch probe status/TP1 Enable
//     Lift1_Enc/Inputs/Lift1_Enc_In/nState6 <-> FB Touch probe status/Touch probe status/TP2 Enable
//     Lift1_Enc/Inputs/Lift1_Enc_In/nState5 @bit 7 <-> FB Touch probe status/Touch probe status/TP1 Input
//     Lift1_Enc/Inputs/Lift1_Enc_In/nState6 @bit 7 <-> FB Touch probe status/Touch probe status/TP2 Input
//     Lift1_Enc/Inputs/Lift1_Enc_In/nState5 @bit 2 <-> FB Touch probe status/Touch probe status/TP1 Neg value stored
//     Lift1_Enc/Inputs/Lift1_Enc_In/nState6 @bit 2 <-> FB Touch probe status/Touch probe status/TP2 Neg value stored
//     Lift1_Enc/Inputs/Lift1_Enc_In/nState5 @bit 1 <-> FB Touch probe status/Touch probe status/TP1 Pos value stored
//     Lift1_Enc/Inputs/Lift1_Enc_In/nState6 @bit 1 <-> FB Touch probe status/Touch probe status/TP2 Pos value stored
//   NC-Task 1 SAF/Axes/Lift2 <-> Device 2 (EtherCAT)/A22.A (Term IO)/A31.2 (Lf2CmdMotor)
//     Lift2_Drive/Inputs/Lift2_Drive_In/nDcOutputTime <-> InfoData/DcOutputShift
//     Lift2_Drive/Inputs/Lift2_Drive_In/nState1 <-> DRV Statusword/Statusword
//     Lift2_Drive/Inputs/Lift2_Drive_In/nState2 <-> DRV Statusword/Statusword @bit 8
//     Lift2_Drive/Inputs/Lift2_Drive_In/nState4 @bit 1 <-> WcState/InputToggle
//     Lift2_Drive/Inputs/Lift2_Drive_In/nState4 <-> WcState/WcState
//     Lift2_Drive/Outputs/Lift2_Drive_Out/nCtrl1 <-> DRV Controlword/Controlword
//     Lift2_Drive/Outputs/Lift2_Drive_Out/nCtrl2 <-> DRV Controlword/Controlword @bit 8
//     Lift2_Drive/Outputs/Lift2_Drive_Out/nDataOut2 <-> DRV Target velocity/Target velocity
//     Lift2_Enc/Inputs/Lift2_Enc_In/nDataIn1 <-> FB Position/Position
//     Lift2_Enc/Inputs/Lift2_Enc_In/nDcInputTime <-> InfoData/DcInputShift
//     Lift2_Enc/Inputs/Lift2_Enc_In/nState4 @bit 1 <-> WcState/InputToggle
//     Lift2_Enc/Inputs/Lift2_Enc_In/nState4 <-> WcState/WcState
//     Lift2_Enc/Inputs/Lift2_Enc_In/nState5 <-> FB Touch probe status/Touch probe status/TP1 Enable
//     Lift2_Enc/Inputs/Lift2_Enc_In/nState6 <-> FB Touch probe status/Touch probe status/TP2 Enable
//     Lift2_Enc/Inputs/Lift2_Enc_In/nState5 @bit 2 <-> FB Touch probe status/Touch probe status/TP1 Neg value stored
//     Lift2_Enc/Inputs/Lift2_Enc_In/nState6 @bit 2 <-> FB Touch probe status/Touch probe status/TP2 Neg value stored
//     Lift2_Enc/Inputs/Lift2_Enc_In/nState5 @bit 1 <-> FB Touch probe status/Touch probe status/TP1 Pos value stored
//     Lift2_Enc/Inputs/Lift2_Enc_In/nState6 @bit 1 <-> FB Touch probe status/Touch probe status/TP2 Pos value stored
//     Lift2_Enc/Inputs/Lift2_Enc_In/nState6 @bit 7 <-> FB Touch probe status/Touch probe status/TP2 Input
//   NC-Task 1 SAF/Axes/Loader Theta <-> Device 2 (EtherCAT)/A22.A (Term IO)/A33.3 (PoAtCmdMotor)
//     Loader Theta_Drive/Inputs/Loader Theta_Drive_In/nState1 @bit 3 <-> STM Status/Status/Error
//     Loader Theta_Drive/Inputs/Loader Theta_Drive_In/nState1 @bit 7 <-> STM Status/Status/Motor stall
//     Loader Theta_Drive/Inputs/Loader Theta_Drive_In/nState1 @bit 5 <-> STM Status/Status/Moving negative
//     Loader Theta_Drive/Inputs/Loader Theta_Drive_In/nState1 @bit 4 <-> STM Status/Status/Moving positive
//     Loader Theta_Drive/Inputs/Loader Theta_Drive_In/nState1 @bit 1 <-> STM Status/Status/Ready
//     Loader Theta_Drive/Inputs/Loader Theta_Drive_In/nState1 <-> STM Status/Status/Ready to enable
//     Loader Theta_Drive/Inputs/Loader Theta_Drive_In/nState1 @bit 6 <-> STM Status/Status/Torque reduced
//     Loader Theta_Drive/Inputs/Loader Theta_Drive_In/nState1 @bit 2 <-> STM Status/Status/Warning
//     Loader Theta_Drive/Inputs/Loader Theta_Drive_In/nState2 @bit 3 <-> STM Status/Status/Digital input 1
//     Loader Theta_Drive/Inputs/Loader Theta_Drive_In/nState2 @bit 4 <-> STM Status/Status/Digital input 2
//     Loader Theta_Drive/Inputs/Loader Theta_Drive_In/nState2 @bit 5 <-> STM Status/Status/Sync error
//     Loader Theta_Drive/Inputs/Loader Theta_Drive_In/nState2 @bit 7 <-> STM Status/Status/TxPDO Toggle
//     Loader Theta_Drive/Inputs/Loader Theta_Drive_In/nState4 @bit 1 <-> WcState/InputToggle
//     Loader Theta_Drive/Inputs/Loader Theta_Drive_In/nState4 <-> WcState/WcState
//     Loader Theta_Drive/Outputs/Loader Theta_Drive_Out/nCtrl1 <-> STM Control/Control/Enable
//     Loader Theta_Drive/Outputs/Loader Theta_Drive_Out/nCtrl1 @bit 2 <-> STM Control/Control/Reduce torque
//     Loader Theta_Drive/Outputs/Loader Theta_Drive_Out/nCtrl1 @bit 1 <-> STM Control/Control/Reset
//     Loader Theta_Drive/Outputs/Loader Theta_Drive_Out/nCtrl2 @bit 3 <-> STM Control/Control/Digital output 1
//     Loader Theta_Drive/Outputs/Loader Theta_Drive_Out/nDataOut2[0] <-> STM Velocity/Velocity
//     Loader Theta_Enc/Inputs/Loader Theta_Enc_In/nDataIn1[0] <-> ENC Status compact/Counter value
//     Loader Theta_Enc/Inputs/Loader Theta_Enc_In/nDataIn2[0] <-> ENC Status compact/Latch value
//     Loader Theta_Enc/Inputs/Loader Theta_Enc_In/nState1 @bit 4 <-> ENC Status compact/Status/Counter overflow
//     Loader Theta_Enc/Inputs/Loader Theta_Enc_In/nState1 @bit 3 <-> ENC Status compact/Status/Counter underflow
//     Loader Theta_Enc/Inputs/Loader Theta_Enc_In/nState1 @bit 7 <-> ENC Status compact/Status/Extrapolation stall
//     Loader Theta_Enc/Inputs/Loader Theta_Enc_In/nState1 <-> ENC Status compact/Status/Latch C valid
//     Loader Theta_Enc/Inputs/Loader Theta_Enc_In/nState1 @bit 1 <-> ENC Status compact/Status/Latch extern valid
//     Loader Theta_Enc/Inputs/Loader Theta_Enc_In/nState1 @bit 2 <-> ENC Status compact/Status/Set counter done
//     Loader Theta_Enc/Inputs/Loader Theta_Enc_In/nState2 @bit 4 <-> ENC Status compact/Status/Status of extern latch
//     Loader Theta_Enc/Inputs/Loader Theta_Enc_In/nState2 <-> ENC Status compact/Status/Status of input A
//     Loader Theta_Enc/Inputs/Loader Theta_Enc_In/nState2 @bit 1 <-> ENC Status compact/Status/Status of input B
//     Loader Theta_Enc/Inputs/Loader Theta_Enc_In/nState2 @bit 2 <-> ENC Status compact/Status/Status of input C
//     Loader Theta_Enc/Inputs/Loader Theta_Enc_In/nState2 @bit 5 <-> ENC Status compact/Status/Sync error
//     Loader Theta_Enc/Inputs/Loader Theta_Enc_In/nState2 @bit 7 <-> ENC Status compact/Status/TxPDO Toggle
//     Loader Theta_Enc/Inputs/Loader Theta_Enc_In/nState4 @bit 1 <-> WcState/InputToggle
//     Loader Theta_Enc/Inputs/Loader Theta_Enc_In/nState4 <-> WcState/WcState
//     Loader Theta_Enc/Outputs/Loader Theta_Enc_Out/nCtrl1 <-> ENC Control compact/Control/Enable latch C
//     Loader Theta_Enc/Outputs/Loader Theta_Enc_Out/nCtrl1 @bit 3 <-> ENC Control compact/Control/Enable latch extern on negative edge
//     Loader Theta_Enc/Outputs/Loader Theta_Enc_Out/nCtrl1 @bit 1 <-> ENC Control compact/Control/Enable latch extern on positive edge
//     Loader Theta_Enc/Outputs/Loader Theta_Enc_Out/nCtrl1 @bit 2 <-> ENC Control compact/Control/Set counter
//     Loader Theta_Enc/Outputs/Loader Theta_Enc_Out/nDataOut1[0] <-> ENC Control compact/Set counter value
//   NC-Task 1 SAF/Axes/Loader X <-> Device 2 (EtherCAT)/A18.2 (PoAxMotor PoAyMotor)
//     Loader X_Drive/Inputs/Loader X_Drive_In/nDataIn1 <-> AT 1/Following distance
//     Loader X_Drive/Inputs/Loader X_Drive_In/nDcOutputTime <-> InfoData/DcOutputShift
//     Loader X_Drive/Inputs/Loader X_Drive_In/nState1 <-> AT 1/Drive status word @bit 8
//     Loader X_Drive/Inputs/Loader X_Drive_In/nState2 <-> AT 1/Drive status word
//     Loader X_Drive/Inputs/Loader X_Drive_In/nState4 @bit 1 <-> WcState/InputToggle
//     Loader X_Drive/Inputs/Loader X_Drive_In/nState4 <-> WcState/WcState
//     Loader X_Drive/Outputs/Loader X_Drive_Out/nCtrl1 <-> MDT 1/Master control word @bit 8
//     Loader X_Drive/Outputs/Loader X_Drive_Out/nDataOut1 <-> MDT 1/Position command value
//     Loader X_Enc/Inputs/Loader X_Enc_In/nDataIn1 <-> AT 1/Position feedback 1 value
//     Loader X_Enc/Inputs/Loader X_Enc_In/nDcInputTime <-> InfoData/DcInputShift
//     Loader X_Enc/Inputs/Loader X_Enc_In/nState4 @bit 1 <-> WcState/InputToggle
//     Loader X_Enc/Inputs/Loader X_Enc_In/nState4 <-> WcState/WcState
//   NC-Task 1 SAF/Axes/Loader Y <-> Device 2 (EtherCAT)/A18.2 (PoAxMotor PoAyMotor)
//     Loader Y_Drive/Inputs/Loader Y_Drive_In/nDataIn1 <-> AT 2/Following distance
//     Loader Y_Drive/Inputs/Loader Y_Drive_In/nDcOutputTime <-> InfoData/DcOutputShift
//     Loader Y_Drive/Inputs/Loader Y_Drive_In/nState1 <-> AT 2/Drive status word @bit 8
//     Loader Y_Drive/Inputs/Loader Y_Drive_In/nState2 <-> AT 2/Drive status word
//     Loader Y_Drive/Inputs/Loader Y_Drive_In/nState4 @bit 1 <-> WcState/InputToggle
//     Loader Y_Drive/Inputs/Loader Y_Drive_In/nState4 <-> WcState/WcState
//     Loader Y_Drive/Outputs/Loader Y_Drive_Out/nCtrl1 <-> MDT 2/Master control word @bit 8
//     Loader Y_Drive/Outputs/Loader Y_Drive_Out/nDataOut1 <-> MDT 2/Position command value
//     Loader Y_Enc/Inputs/Loader Y_Enc_In/nDataIn1 <-> AT 2/Position feedback 1 value
//     Loader Y_Enc/Inputs/Loader Y_Enc_In/nDcInputTime <-> InfoData/DcInputShift
//     Loader Y_Enc/Inputs/Loader Y_Enc_In/nState4 @bit 1 <-> WcState/InputToggle
//     Loader Y_Enc/Inputs/Loader Y_Enc_In/nState4 <-> WcState/WcState
//   NC-Task 1 SAF/Axes/Loader Z1 <-> Device 2 (EtherCAT)/A22.A (Term IO)/A33.1 (PoAz1MotCmd)
//     Drive/Inputs/In/nDcOutputTime <-> InfoData/DcOutputShift
//     Drive/Inputs/In/nState1 <-> DRV Statusword/Statusword
//     Drive/Inputs/In/nState2 <-> DRV Statusword/Statusword @bit 8
//     Drive/Inputs/In/nState4 @bit 1 <-> WcState/InputToggle
//     Drive/Inputs/In/nState4 <-> WcState/WcState
//     Drive/Outputs/Out/nCtrl1 <-> DRV Controlword/Controlword
//     Drive/Outputs/Out/nCtrl2 <-> DRV Controlword/Controlword @bit 8
//     Drive/Outputs/Out/nDataOut2 <-> DRV Target velocity/Target velocity
//     Enc/Inputs/In/nDataIn1 <-> FB Position/Position
//     Enc/Inputs/In/nDcInputTime <-> InfoData/DcInputShift
//     Enc/Inputs/In/nState4 @bit 1 <-> WcState/InputToggle
//     Enc/Inputs/In/nState4 <-> WcState/WcState
//   NC-Task 1 SAF/Axes/Loader Z2 <-> Device 2 (EtherCAT)/A22.A (Term IO)/A33.2 (PoAz2MotCmd)
//     Drive/Inputs/In/nDcOutputTime <-> InfoData/DcOutputShift
//     Drive/Inputs/In/nState1 <-> DRV Statusword/Statusword
//     Drive/Inputs/In/nState2 <-> DRV Statusword/Statusword @bit 8
//     Drive/Inputs/In/nState4 @bit 1 <-> WcState/InputToggle
//     Drive/Inputs/In/nState4 <-> WcState/WcState
//     Drive/Outputs/Out/nCtrl1 <-> DRV Controlword/Controlword
//     Drive/Outputs/Out/nCtrl2 <-> DRV Controlword/Controlword @bit 8
//     Drive/Outputs/Out/nDataOut2 <-> DRV Target velocity/Target velocity
//     Enc/Inputs/In/nDataIn1 <-> FB Position/Position
//     Enc/Inputs/In/nDcInputTime <-> InfoData/DcInputShift
//     Enc/Inputs/In/nState4 @bit 1 <-> WcState/InputToggle
//     Enc/Inputs/In/nState4 <-> WcState/WcState
//   NC-Task 1 SAF/Axes/Pearling X <-> Device 2 (EtherCAT)/A18.1 (PeAxMotor PeAyMotor)
//     Pearling X_Drive/Inputs/Pearling X_Drive_In/nDataIn1 <-> AT 1/Following distance
//     Pearling X_Drive/Inputs/Pearling X_Drive_In/nDcOutputTime <-> InfoData/DcOutputShift
//     Pearling X_Drive/Inputs/Pearling X_Drive_In/nState1 <-> AT 1/Drive status word @bit 8
//     Pearling X_Drive/Inputs/Pearling X_Drive_In/nState2 <-> AT 1/Drive status word
//     Pearling X_Drive/Inputs/Pearling X_Drive_In/nState4 @bit 1 <-> WcState/InputToggle
//     Pearling X_Drive/Inputs/Pearling X_Drive_In/nState4 <-> WcState/WcState
//     Pearling X_Drive/Outputs/Pearling X_Drive_Out/nCtrl1 <-> MDT 1/Master control word @bit 8
//     Pearling X_Drive/Outputs/Pearling X_Drive_Out/nDataOut1 <-> MDT 1/Position command value
//     Pearling X_Enc/Inputs/Pearling X_Enc_In/nDataIn1 <-> AT 1/Position feedback 1 value
//     Pearling X_Enc/Inputs/Pearling X_Enc_In/nDcInputTime <-> InfoData/DcInputShift
//     Pearling X_Enc/Inputs/Pearling X_Enc_In/nState4 @bit 1 <-> WcState/InputToggle
//     Pearling X_Enc/Inputs/Pearling X_Enc_In/nState4 <-> WcState/WcState
//   NC-Task 1 SAF/Axes/Pearling Y <-> Device 2 (EtherCAT)/A18.1 (PeAxMotor PeAyMotor)
//     Pearling Y_Drive/Inputs/Pearling Y_Drive_In/nDataIn1 <-> AT 2/Following distance
//     Pearling Y_Drive/Inputs/Pearling Y_Drive_In/nDcOutputTime <-> InfoData/DcOutputShift
//     Pearling Y_Drive/Inputs/Pearling Y_Drive_In/nState1 <-> AT 2/Drive status word @bit 8
//     Pearling Y_Drive/Inputs/Pearling Y_Drive_In/nState2 <-> AT 2/Drive status word
//     Pearling Y_Drive/Inputs/Pearling Y_Drive_In/nState4 @bit 1 <-> WcState/InputToggle
//     Pearling Y_Drive/Inputs/Pearling Y_Drive_In/nState4 <-> WcState/WcState
//     Pearling Y_Drive/Outputs/Pearling Y_Drive_Out/nCtrl1 <-> MDT 2/Master control word @bit 8
//     Pearling Y_Drive/Outputs/Pearling Y_Drive_Out/nDataOut1 <-> MDT 2/Position command value
//     Pearling Y_Enc/Inputs/Pearling Y_Enc_In/nDataIn1 <-> AT 2/Position feedback 1 value
//     Pearling Y_Enc/Inputs/Pearling Y_Enc_In/nDcInputTime <-> InfoData/DcInputShift
//     Pearling Y_Enc/Inputs/Pearling Y_Enc_In/nState4 @bit 1 <-> WcState/InputToggle
//     Pearling Y_Enc/Inputs/Pearling Y_Enc_In/nState4 <-> WcState/WcState
//   NC-Task 1 SAF/Axes/Pearling Z1 <-> Device 2 (EtherCAT)/A22.A (Term IO)/A31.3 (PeZ1CmdMotor)
//     Drive/Inputs/In/nDcOutputTime <-> InfoData/DcOutputShift
//     Drive/Inputs/In/nState1 <-> DRV Statusword/Statusword
//     Drive/Inputs/In/nState2 <-> DRV Statusword/Statusword @bit 8
//     Drive/Inputs/In/nState4 @bit 1 <-> WcState/InputToggle
//     Drive/Inputs/In/nState4 <-> WcState/WcState
//     Drive/Outputs/Out/nCtrl1 <-> DRV Controlword/Controlword
//     Drive/Outputs/Out/nCtrl2 <-> DRV Controlword/Controlword @bit 8
//     Drive/Outputs/Out/nDataOut2 <-> DRV Target velocity/Target velocity
//     Enc/Inputs/In/nDataIn1 <-> FB Position/Position
//     Enc/Inputs/In/nDcInputTime <-> InfoData/DcInputShift
//     Enc/Inputs/In/nState4 @bit 1 <-> WcState/InputToggle
//     Enc/Inputs/In/nState4 <-> WcState/WcState
//   NC-Task 1 SAF/Axes/Pearling Z2 <-> Device 2 (EtherCAT)/A22.A (Term IO)/A31.4 (PeZ2CmdMotor)
//     Drive/Inputs/In/nDcOutputTime <-> InfoData/DcOutputShift
//     Drive/Inputs/In/nState1 <-> DRV Statusword/Statusword
//     Drive/Inputs/In/nState2 <-> DRV Statusword/Statusword @bit 8
//     Drive/Inputs/In/nState4 @bit 1 <-> WcState/InputToggle
//     Drive/Inputs/In/nState4 <-> WcState/WcState
//     Drive/Outputs/Out/nCtrl1 <-> DRV Controlword/Controlword
//     Drive/Outputs/Out/nCtrl2 <-> DRV Controlword/Controlword @bit 8
//     Drive/Outputs/Out/nDataOut2 <-> DRV Target velocity/Target velocity
//     Enc/Inputs/In/nDataIn1 <-> FB Position/Position
//     Enc/Inputs/In/nDcInputTime <-> InfoData/DcInputShift
//     Enc/Inputs/In/nState4 @bit 1 <-> WcState/InputToggle
//     Enc/Inputs/In/nState4 <-> WcState/WcState
//   NC-Task 1 SAF/Axes/Sharpen <-> Device 2 (EtherCAT)/A22.A (Term IO)/A34.1 (ShCmdMotor)
//     Sharpen_Drive/Inputs/Sharpen_Drive_In/nDcOutputTime <-> InfoData/DcOutputShift
//     Sharpen_Drive/Inputs/Sharpen_Drive_In/nState1 @bit 3 <-> STM Status/Status/Error
//     Sharpen_Drive/Inputs/Sharpen_Drive_In/nState1 @bit 7 <-> STM Status/Status/Motor stall
//     Sharpen_Drive/Inputs/Sharpen_Drive_In/nState1 @bit 5 <-> STM Status/Status/Moving negative
//     Sharpen_Drive/Inputs/Sharpen_Drive_In/nState1 @bit 4 <-> STM Status/Status/Moving positive
//     Sharpen_Drive/Inputs/Sharpen_Drive_In/nState1 @bit 1 <-> STM Status/Status/Ready
//     Sharpen_Drive/Inputs/Sharpen_Drive_In/nState1 <-> STM Status/Status/Ready to enable
//     Sharpen_Drive/Inputs/Sharpen_Drive_In/nState1 @bit 6 <-> STM Status/Status/Torque reduced
//     Sharpen_Drive/Inputs/Sharpen_Drive_In/nState1 @bit 2 <-> STM Status/Status/Warning
//     Sharpen_Drive/Inputs/Sharpen_Drive_In/nState2 @bit 3 <-> STM Status/Status/Digital input 1
//     Sharpen_Drive/Inputs/Sharpen_Drive_In/nState2 @bit 4 <-> STM Status/Status/Digital input 2
//     Sharpen_Drive/Inputs/Sharpen_Drive_In/nState2 @bit 5 <-> STM Status/Status/Sync error
//     Sharpen_Drive/Inputs/Sharpen_Drive_In/nState2 @bit 7 <-> STM Status/Status/TxPDO Toggle
//     Sharpen_Drive/Inputs/Sharpen_Drive_In/nState4 @bit 1 <-> WcState/InputToggle
//     Sharpen_Drive/Inputs/Sharpen_Drive_In/nState4 <-> WcState/WcState
//     Sharpen_Drive/Outputs/Sharpen_Drive_Out/nCtrl1 <-> STM Control/Control/Enable
//     Sharpen_Drive/Outputs/Sharpen_Drive_Out/nCtrl1 @bit 2 <-> STM Control/Control/Reduce torque
//     Sharpen_Drive/Outputs/Sharpen_Drive_Out/nCtrl1 @bit 1 <-> STM Control/Control/Reset
//     Sharpen_Drive/Outputs/Sharpen_Drive_Out/nCtrl2 @bit 3 <-> STM Control/Control/Digital output 1
//     Sharpen_Drive/Outputs/Sharpen_Drive_Out/nDataOut2[0] <-> STM Velocity/Velocity
//   NC-Task 1 SAF/Axes/SharpenEncoder <-> Device 2 (EtherCAT)/A22.A (Term IO)/A34.1 (ShCmdMotor)
//     SharpenEncoder_Enc/Inputs/SharpenEncoder_Enc_In/nDataIn1[0] <-> ENC Status compact/Counter value
//     SharpenEncoder_Enc/Inputs/SharpenEncoder_Enc_In/nDataIn2[0] <-> ENC Status compact/Latch value
//     SharpenEncoder_Enc/Inputs/SharpenEncoder_Enc_In/nDcInputTime <-> InfoData/DcInputShift
//     SharpenEncoder_Enc/Inputs/SharpenEncoder_Enc_In/nState1 @bit 4 <-> ENC Status compact/Status/Counter overflow
//     SharpenEncoder_Enc/Inputs/SharpenEncoder_Enc_In/nState1 @bit 3 <-> ENC Status compact/Status/Counter underflow
//     SharpenEncoder_Enc/Inputs/SharpenEncoder_Enc_In/nState1 @bit 7 <-> ENC Status compact/Status/Extrapolation stall
//     SharpenEncoder_Enc/Inputs/SharpenEncoder_Enc_In/nState1 <-> ENC Status compact/Status/Latch C valid
//     SharpenEncoder_Enc/Inputs/SharpenEncoder_Enc_In/nState1 @bit 1 <-> ENC Status compact/Status/Latch extern valid
//     SharpenEncoder_Enc/Inputs/SharpenEncoder_Enc_In/nState1 @bit 2 <-> ENC Status compact/Status/Set counter done
//     SharpenEncoder_Enc/Inputs/SharpenEncoder_Enc_In/nState2 @bit 4 <-> ENC Status compact/Status/Status of extern latch
//     SharpenEncoder_Enc/Inputs/SharpenEncoder_Enc_In/nState2 <-> ENC Status compact/Status/Status of input A
//     SharpenEncoder_Enc/Inputs/SharpenEncoder_Enc_In/nState2 @bit 1 <-> ENC Status compact/Status/Status of input B
//     SharpenEncoder_Enc/Inputs/SharpenEncoder_Enc_In/nState2 @bit 2 <-> ENC Status compact/Status/Status of input C
//     SharpenEncoder_Enc/Inputs/SharpenEncoder_Enc_In/nState2 @bit 5 <-> ENC Status compact/Status/Sync error
//     SharpenEncoder_Enc/Inputs/SharpenEncoder_Enc_In/nState2 @bit 7 <-> ENC Status compact/Status/TxPDO Toggle
//     SharpenEncoder_Enc/Inputs/SharpenEncoder_Enc_In/nState4 @bit 1 <-> WcState/InputToggle
//     SharpenEncoder_Enc/Inputs/SharpenEncoder_Enc_In/nState4 <-> WcState/WcState
//     SharpenEncoder_Enc/Outputs/SharpenEncoder_Enc_Out/nCtrl1 <-> ENC Control compact/Control/Enable latch C
//     SharpenEncoder_Enc/Outputs/SharpenEncoder_Enc_Out/nCtrl1 @bit 3 <-> ENC Control compact/Control/Enable latch extern on negative edge
//     SharpenEncoder_Enc/Outputs/SharpenEncoder_Enc_Out/nCtrl1 @bit 1 <-> ENC Control compact/Control/Enable latch extern on positive edge
//     SharpenEncoder_Enc/Outputs/SharpenEncoder_Enc_Out/nCtrl1 @bit 2 <-> ENC Control compact/Control/Set counter
//     SharpenEncoder_Enc/Outputs/SharpenEncoder_Enc_Out/nDataOut1[0] <-> ENC Control compact/Set counter value
//   NC-Task 1 SAF/Axes/Table <-> Device 2 (EtherCAT)/A18.3 Table (AX5203-0000-0203)
//     Table_Drive/Inputs/Table_Drive_In/nDataIn1 <-> AT 1/Following distance
//     Table_Drive/Inputs/Table_Drive_In/nDcOutputTime <-> InfoData/DcOutputShift
//     Table_Drive/Inputs/Table_Drive_In/nState1 <-> AT 1/Drive status word @bit 8
//     Table_Drive/Inputs/Table_Drive_In/nState2 <-> AT 1/Drive status word
//     Table_Drive/Inputs/Table_Drive_In/nState4 @bit 1 <-> WcState/InputToggle
//     Table_Drive/Inputs/Table_Drive_In/nState4 <-> WcState/WcState
//     Table_Drive/Outputs/Table_Drive_Out/nCtrl1 <-> MDT 1/Master control word @bit 8
//     Table_Drive/Outputs/Table_Drive_Out/nDataOut1 <-> MDT 1/Position command value
//     Table_Enc/Inputs/Table_Enc_In/nDataIn1 <-> AT 1/Position feedback 1 value
//     Table_Enc/Inputs/Table_Enc_In/nDcInputTime <-> InfoData/DcInputShift
//     Table_Enc/Inputs/Table_Enc_In/nState4 @bit 1 <-> WcState/InputToggle
//     Table_Enc/Inputs/Table_Enc_In/nState4 <-> WcState/WcState
//   Perlage_Standard/Perlage_Standard Instance <-> Device 2 (EtherCAT)/A18.1 (PeAxMotor PeAyMotor)
//     Standard Inputs/.IPearlingMotorXYStatus <-> AT 1/Digital inputs, state
//   Perlage_Standard/Perlage_Standard Instance <-> Device 2 (EtherCAT)/A18.2 (PoAxMotor PoAyMotor)
//     Standard Inputs/.ILoaderMotorXYStatus <-> AT 1/Digital inputs, state
//   Perlage_Standard/Perlage_Standard Instance <-> Device 2 (EtherCAT)/A18.3 Table (AX5203-0000-0203)
//     Standard Inputs/.IbTableHome <-> AT 1/Digital inputs, state
//   Perlage_Standard/Perlage_Standard Instance <-> Device 2 (EtherCAT)/A22.A (Term IO)/A22.1
//     Standard Inputs/.Ib24VOK <-> Channel 1/Supply24VOn
//     Standard Inputs/.Ib48VOK <-> Channel 2/Supply48VOn
//     Standard Inputs/.IbAirPressureOK <-> Channel 3/AirSupplyOk
//     Standard Inputs/.IbLift1DrawerInPos <-> Channel 12/Lf1DrawInPos
//     Standard Inputs/.IbLift1NegLimit <-> Channel 9/Lf1LimiteDown
//     Standard Inputs/.IbLift2NegLimit <-> Channel 13/Lf2LimiteDown
//     Standard Inputs/.IbLift1PlateInPos <-> Channel 11/Lf1PlatelnPos
//     Standard Inputs/.IbLift2PlateInPos <-> Channel 15/Lf2PlatelnPos
//     Standard Inputs/.IbLift1PosLimit <-> Channel 10/Lf1LimiteUp
//     Standard Inputs/.IbLift2PosLimit <-> Channel 14/Lf2LimiteUp
//     Standard Inputs/.IbLift2DrawerInPos <-> Channel 16/Lf2DrawlnPos
//     Standard Inputs/.IbMainVacuumOK <-> Channel 7/VacPumpPressureOk
//     Standard Inputs/.IbPearlingChangeBroach <-> Channel 4/PeSeqChangSpin
//     Standard Inputs/.IbVacuumPumpIsOn <-> Channel 6/VacuumPumpIsOn
//   Perlage_Standard/Perlage_Standard Instance <-> Device 2 (EtherCAT)/A22.A (Term IO)/A22.2
//     Standard Inputs/.IbAspirationIsOn <-> Channel 1/VacuCleanRFiltrOk
//     Standard Inputs/.IbAspirationOK <-> Channel 2/VacCleanFlowOk
//     Standard Inputs/.IbLoaderHomeZ1 <-> Channel 3/PoAz1IsHome
//     Standard Inputs/.IbLoaderHomeZ2 <-> Channel 4/PoAz2IsHome
//     Standard Inputs/.IbLoaderNegLimitZ1 <-> Channel 8/PoAz1LimiteUp
//     Standard Inputs/.IbLoaderNegLimitZ2 <-> Channel 11/PoAz2LimiteUp
//     Standard Inputs/.IbLoaderPlateTakerIsDown <-> Channel 14/PoTakPalDown
//     Standard Inputs/.IbLoaderPlateTakerIsUp <-> Channel 13/PoTakPalUp
//     Standard Inputs/.IbLoaderPlateVacuumOK <-> Channel 15/PoTakPlaVacOK
//     Standard Inputs/.IbLoaderPosLimitZ1 <-> Channel 7/PoAz1LimiteDown
//     Standard Inputs/.IbLoaderPosLimitZ2 <-> Channel 10/PoAz2LimiteDown
//     Standard Inputs/.IbRejectDrawerInPos <-> Channel 6/RjDrawerlnPos
//     Standard Inputs/.IbRejectPlateInPos <-> Channel 5/RjPlatelnPos
//   Perlage_Standard/Perlage_Standard Instance <-> Device 2 (EtherCAT)/A22.A (Term IO)/A22.3
//     Standard Inputs/.IbPearlingChuck1Closed <-> Channel 9/SpZ1GripIsClosed
//     Standard Inputs/.IbPearlingChuck2Closed <-> Channel 7/SpZ2GripIsClosed
//     Standard Inputs/.IbPearlingChuck1Open <-> Channel 10/SpZ1GripIsOpen
//     Standard Inputs/.IbPearlingChuck2Open <-> Channel 8/SpZ2GripIsOpen
//     Standard Inputs/.IbPearlingHomeZ1 <-> Channel 1/PeZ1AzIsHome
//     Standard Inputs/.IbPearlingHomeZ2 <-> Channel 4/PeZ2AzIsHome
//     Standard Inputs/.IbPearlingNegLimitZ1 <-> Channel 2/PeZ1AzLimitUp
//     Standard Inputs/.IbPearlingNegLimitZ2 <-> Channel 5/PeZ2AzLimitUp
//     Standard Inputs/.IbPearlingPosLimitZ1 <-> Channel 3/PeZ1AzLimitDown
//     Standard Inputs/.IbPearlingPosLimitZ2 <-> Channel 6/PeZ2AzLimitDown
//     Standard Inputs/.IbTableAspirationIsDown <-> Channel 16/RtSpinAspIsDown
//     Standard Inputs/.IbTableAspirationIsUp <-> Channel 15/RtSpAspIsUp
//     Standard Inputs/.IbTableCleanBrushIsDown <-> Channel 12/BrosseBas
//     Standard Inputs/.IbTableCleanBrushIsUp <-> Channel 11/BrosseHaut
//     Standard Inputs/.IbTableLocked <-> Channel 13/Rtlndexed
//     Standard Inputs/.IbTableNotLocked <-> Channel 14/RtUnindexed
//   Perlage_Standard/Perlage_Standard Instance <-> Device 2 (EtherCAT)/A22.A (Term IO)/A22.4
//     Standard Inputs/.IbBarrelIndexed <-> Channel 8/Balndexed
//     Standard Inputs/.IbBarrelNotIndexed <-> Channel 9/ClNotIndexed
//     Standard Inputs/.IbBarrelStickIsDown <-> Channel 10/ClSticklsDown
//     Standard Inputs/.IbBarrelStickIsUp <-> Channel 11/ClSticklsUp
//     Standard Inputs/.IbBarrelStickPresent <-> Channel 12/ClSticklsPres
//     Standard Inputs/.IbBrushHome <-> Channel 13/BrHomePos
//     Standard Inputs/.IbBrushNegLimit <-> Channel 14/BrLimiit-
//     Standard Inputs/.IbBrushPosLimit <-> Channel 15/BrLimit+
//     Standard Inputs/.IbSharpenPosTensioner <-> Channel 7/ShCtrlPosTend
//     Standard Inputs/.IbTurnOverFixIsDown <-> Channel 3/RelsDown
//     Standard Inputs/.IbTurnOverFixIsUp <-> Channel 4/RelsUp
//   Perlage_Standard/Perlage_Standard Instance <-> Device 2 (EtherCAT)/A22.A (Term IO)/A23.1
//     Standard Inputs/.IbLift1DrawerLocked <-> Channel 3/Drawer1Locked
//     Standard Inputs/.IbLift2DrawerLocked <-> Channel 7/Drawer2Locked
//     Standard Inputs/.IbLift1DrawerUnlocked <-> Channel 4/Drawer1Unlocked
//     Standard Inputs/.IbLift2DrawerUnlocked <-> Channel 8/Drawer2Unlocked
//     Standard Inputs/.IbLift1PlateLocked <-> Channel 1/Plate1Locked
//     Standard Inputs/.IbLift2PlateLocked <-> Channel 5/Plate2Locked
//     Standard Inputs/.IbLift1PlateUnlocked <-> Channel 2/Plate1Unlocked
//     Standard Inputs/.IbLift2PlateUnlocked <-> Channel 6/Plate2Unlocked
//   Perlage_Standard/Perlage_Standard Instance <-> Device 2 (EtherCAT)/A22.A (Term IO)/A25.1
//     Standard Inputs/.ILoaderPlateDistance <-> AI Standard Channel 1/PoTrayHeigMeas
//     Standard Inputs/.IPearlingContact1Distance <-> AI Standard Channel 3/PeZ1AzPresCtrl
//     Standard Inputs/.IPearlingContact2Distance <-> AI Standard Channel 2/PeZ2AzPresCtrl
//   Perlage_Standard/Perlage_Standard Instance <-> Device 2 (EtherCAT)/A22.A (Term IO)/A25.2
//     Standard Inputs/.IiTableVacuumPos{1..4}Flow <-> AI Standard Channel {1..4}/RtLayring{1..4}Vac  (4 links)
//   Perlage_Standard/Perlage_Standard Instance <-> Device 2 (EtherCAT)/A22.A (Term IO)/A25.3
//     Standard Inputs/.IPearlingWeightMeasure <-> AI Standard Channel 1/CaLoadSensor
//   Perlage_Standard/Perlage_Standard Instance <-> Device 2 (EtherCAT)/A22.A (Term IO)/A25.4
//     Standard Inputs/.IiLoaderHead1Vacuum <-> AI Standard Channel 2/PoAz1VacOK
//     Standard Inputs/.IiLoaderHead2Vacuum <-> AI Standard Channel 1/PoAz2VacOK
//   Perlage_Standard/Perlage_Standard Instance <-> Device 2 (EtherCAT)/A22.A (Term IO)/A26.1
//     Standard Outputs/.QbLockLoaderDoors <-> Channel 1/Safety1Lock
//     Standard Outputs/.QbLockLoaderDoors <-> Channel 2/Safety2Lock
//     Standard Outputs/.QbLockPearlingDoors <-> Channel 3/Safety3Lock
//     Standard Outputs/.QbLockPearlingDoors <-> Channel 4/Safety4Lock
//   Perlage_Standard/Perlage_Standard Instance <-> Device 2 (EtherCAT)/A22.A (Term IO)/A26.2
//     Standard Outputs/.QbBlueLight <-> Channel 3/BlueLight
//     Standard Outputs/.QbGreenLight <-> Channel 1/GreenLight
//     Standard Outputs/.QbLift1BlueLight <-> Channel 6/Lf1BlueLight
//     Standard Outputs/.QbLift2BlueLight <-> Channel 7/Lf2BlueLight
//     Standard Outputs/.QbLoaderActivateHead1Blowing <-> Channel 15/PoAz1BlowOn
//     Standard Outputs/.QbLoaderActivateHead2Blowing <-> Channel 10/PoAz2BlowOn
//     Standard Outputs/.QbLoaderActivateHead1Vacuum <-> Channel 14/PoAz1VacOn
//     Standard Outputs/.QbLoaderActivateHead2Vacuum <-> Channel 4/PoAz2VacOn
//     Standard Outputs/.QbPearlingChangeBroachLight <-> Channel 11/PeLedSeqChangSp
//     Standard Outputs/.QbPearlingStickLed1 <-> Channel 12/SpZ1LedApp
//     Standard Outputs/.QbPearlingStickLed2 <-> Channel 13/SpZ2LedApp
//     Standard Outputs/.QbRedLight <-> Channel 2/RedLight
//     Standard Outputs/.QbRejectBlueLight <-> Channel 9/RjBlueLight
//     Standard Outputs/.QbVacuumPumpOn <-> Channel 5/CmdVacuumPump
//   Perlage_Standard/Perlage_Standard Instance <-> Device 2 (EtherCAT)/A22.A (Term IO)/A28.1
//     Standard Outputs/.QbAspirationOn <-> Channel 3/VacuCleanRCmd
//     Standard Outputs/.QbPearlingStartMotor1 <-> Channel 2/SpLCtrlMot
//     Standard Outputs/.QbPearlingStartMotor2 <-> Channel 1/SpRCtrlMot
//   Perlage_Standard/Perlage_Standard Instance <-> Device 2 (EtherCAT)/A22.A (Term IO)/A29.1 (Twinsafe PLC)
//     Standard Inputs/.IbLoaderDoorsClosed <-> Device Info Data/Internal I/O/Input Safe Data FSIN Module 3.Input
//     Standard Inputs/.IbLoaderDoorsLocked <-> Device Info Data/Internal I/O/Input Safe Data FSIN Module 4.Input
//     Standard Inputs/.IbNoEmergencyStop <-> Device Info Data/Internal I/O/Input Safe Data FSIN Module 1.Input
//     Standard Inputs/.IbPearlingDoorsClosed <-> Device Info Data/Internal I/O/Input Safe Data FSIN Module 5.Input
//     Standard Inputs/.IbPearlingDoorsLocked <-> Device Info Data/Internal I/O/Input Safe Data FSIN Module 6.Input
//     Standard Outputs/.QbPowerOnDrives <-> StandardOutputs/TwinSafeGroup1.QbPowerOnDrives_11
//     Standard Outputs/.QbResetSafety <-> StandardOutputs/TwinSafeGroup1.QBResetSafety_6
//     Standard Outputs/.QbStartSafety <-> StandardOutputs/TwinSafeGroup1.QBStartSafety_7
//   Perlage_Standard/Perlage_Standard Instance <-> Device 2 (EtherCAT)/A22.A (Term IO)/A29.4 (TwinSafe IN)
//     Standard Inputs/.IbDrivesAreOFF <-> Module 1 (FSOES)/TxPDO/FSOE/DriveIsOn1
//     Standard Inputs/.IbV1PowerIsOff <-> Module 1 (FSOES)/TxPDO/FSOE/PwrV1IsOn_1
//   Perlage_Standard/Perlage_Standard Instance <-> Device 2 (EtherCAT)/A22.A (Term IO)/A31.1 (Lf1CmdMotor)
//     Standard Inputs/.IbLift1Home <-> FB Touch probe status/Touch probe status/TP1 Input
//   Perlage_Standard/Perlage_Standard Instance <-> Device 2 (EtherCAT)/A22.A (Term IO)/A31.2 (Lf2CmdMotor)
//     Standard Inputs/.IbLift2Home <-> FB Touch probe status/Touch probe status/TP1 Input
//   Perlage_Standard/Perlage_Standard Instance <-> Device 2 (EtherCAT)/A22.A (Term IO)/A33.4 (ReCmdMotor)
//     Standard Inputs/.IbTurnOverHome <-> STM Status/Status/Digital input 1
//   Perlage_Standard/Perlage_Standard Instance <-> Device 2 (EtherCAT)/A75.1
//     Standard Outputs/.QbBarrelIndexTable <-> Byte 1/Output[2]
//     Standard Outputs/.QbBarrelMoveUpStick <-> Byte 1/Output[4]
//     Standard Outputs/.QbLift1LockDrawer <-> Byte 2/Output[6]
//     Standard Outputs/.QbLift2LockDrawer <-> Byte 3/Output[2]
//     Standard Outputs/.QbLift1LockPlate <-> Byte 2/Output[4]
//     Standard Outputs/.QbLift2LockPlate <-> Byte 3/Output[0]
//     Standard Outputs/.QbLift1UnlockDrawer <-> Byte 2/Output[7]
//     Standard Outputs/.QbLift2UnlockDrawer <-> Byte 3/Output[3]
//     Standard Outputs/.QbLift1UnlockPlate <-> Byte 2/Output[5]
//     Standard Outputs/.QbLift2UnlockPlate <-> Byte 3/Output[1]
//     Standard Outputs/.QbLoaderPlateTakerDown <-> Byte 2/Output[0]
//     Standard Outputs/.QbLoaderPlateTakerUp <-> Byte 2/Output[1]
//     Standard Outputs/.QbPearlingActivateBlowing1 <-> Byte 0/Output[6]
//     Standard Outputs/.QbPearlingActivateBlowing2 <-> Byte 0/Output[2]
//     Standard Outputs/.QbPearlingActivateEject1 <-> Byte 0/Output[4]
//     Standard Outputs/.QbPearlingActivateEject2 <-> Byte 0/Output[0]
//     Standard Outputs/.QbPearlingOpenChuck1 <-> Byte 3/Output[6]
//     Standard Outputs/.QbPearlingOpenChuck2 <-> Byte 3/Output[4]
//     Standard Outputs/.QbTableAspirationDown <-> Byte 2/Output[2]
//     Standard Outputs/.QbTableAspirationUp <-> Byte 2/Output[3]
//     Standard Outputs/.QbTableCleanBrushDown <-> Byte 1/Output[6]
//     Standard Outputs/.QbTableLock <-> Byte 1/Output[0]
//   Perlage_Standard/Perlage_Standard Instance <-> Device 2 (EtherCAT)/A79.1
//     Standard Outputs/.QbBrushAspirationBlowing <-> Byte 0/Output[2]
//     Standard Outputs/.QbBrushAspirationVacuum <-> Byte 0/Output[3]
//     Standard Outputs/.QbLoaderActivatePlateBlowing <-> Byte 0/Output[0]
//     Standard Outputs/.QbLoaderActivatePlateVacuum <-> Byte 0/Output[1]
//     Standard Outputs/.QbSharpenAspirationBlowing <-> Byte 1/Output[2]
//     Standard Outputs/.QbSharpenAspirationVacuum <-> Byte 1/Output[3]
//     Standard Outputs/.QbTableAspiration13Blowing <-> Byte 0/Output[4]
//     Standard Outputs/.QbTableAspiration24Blowing <-> Byte 0/Output[6]
//     Standard Outputs/.QbTableAspiration13Vacuum <-> Byte 0/Output[5]
//     Standard Outputs/.QbTableAspiration24Vacuum <-> Byte 0/Output[7]
//   Perlage_Standard/Perlage_Standard Instance <-> Device 2 (EtherCAT)/A79.2
//     Standard Outputs/.QbTableActivateBlowingPos{1..4} <-> Byte 0/Output[{0..6 step 2}]  (4 links)
//     Standard Outputs/.QbTableActivateVacuumPos{1..4} <-> Byte 0/Output[{1..7 step 2}]  (4 links)
//   Perlage_Standard/Perlage_Standard Instance <-> NC-Task 1 SAF/Axes/Barrel
//     Standard Inputs/.TBarrelAxis.NcToPlc <-> Outputs/Barrel_ToPlc
//     Standard Outputs/.TBarrelAxis.PlcToNc <-> Inputs/Barrel_FromPlc
//   Perlage_Standard/Perlage_Standard Instance <-> NC-Task 1 SAF/Axes/Brush
//     Standard Inputs/.TBrushAxis.NcToPlc <-> Outputs/Brush_ToPlc
//     Standard Outputs/.TBrushAxis.PlcToNc <-> Inputs/Brush_FromPlc
//   Perlage_Standard/Perlage_Standard Instance <-> NC-Task 1 SAF/Axes/Lift1
//     Standard Inputs/.TLift1Axis.NcToPlc <-> Outputs/Lift1_ToPlc
//     Standard Outputs/.TLift1Axis.PlcToNc <-> Inputs/Lift1_FromPlc
//   Perlage_Standard/Perlage_Standard Instance <-> NC-Task 1 SAF/Axes/Lift2
//     Standard Inputs/.TLift2Axis.NcToPlc <-> Outputs/Lift2_ToPlc
//     Standard Outputs/.TLift2Axis.PlcToNc <-> Inputs/Lift2_FromPlc
//   Perlage_Standard/Perlage_Standard Instance <-> NC-Task 1 SAF/Axes/Loader Theta
//     Standard Inputs/.TLoaderThetaAxis.NcToPlc <-> Outputs/Loader Theta_ToPlc
//     Standard Outputs/.TLoaderThetaAxis.PlcToNc <-> Inputs/Loader Theta_FromPlc
//   Perlage_Standard/Perlage_Standard Instance <-> NC-Task 1 SAF/Axes/Loader X
//     Standard Inputs/.TLoaderXAxis.NcToPlc <-> Outputs/Loader X_ToPlc
//     Standard Outputs/.TLoaderXAxis.PlcToNc <-> Inputs/Loader X_FromPlc
//   Perlage_Standard/Perlage_Standard Instance <-> NC-Task 1 SAF/Axes/Loader Y
//     Standard Inputs/.TLoaderYAxis.NcToPlc <-> Outputs/Loader Y_ToPlc
//     Standard Outputs/.TLoaderYAxis.PlcToNc <-> Inputs/Loader Y_FromPlc
//   Perlage_Standard/Perlage_Standard Instance <-> NC-Task 1 SAF/Axes/Loader Z1
//     Standard Inputs/.TLoaderZ1Axis.NcToPlc <-> Outputs/ToPlc
//     Standard Outputs/.TLoaderZ1Axis.PlcToNc <-> Inputs/FromPlc
//   Perlage_Standard/Perlage_Standard Instance <-> NC-Task 1 SAF/Axes/Loader Z2
//     Standard Inputs/.TLoaderZ2Axis.NcToPlc <-> Outputs/ToPlc
//     Standard Outputs/.TLoaderZ2Axis.PlcToNc <-> Inputs/FromPlc
//   Perlage_Standard/Perlage_Standard Instance <-> NC-Task 1 SAF/Axes/Pearling X
//     Standard Inputs/.TPearlingXAxis.NcToPlc <-> Outputs/Pearling X_ToPlc
//     Standard Outputs/.TPearlingXAxis.PlcToNc <-> Inputs/Pearling X_FromPlc
//   Perlage_Standard/Perlage_Standard Instance <-> NC-Task 1 SAF/Axes/Pearling Y
//     Standard Inputs/.TPearlingYAxis.NcToPlc <-> Outputs/Pearling Y_ToPlc
//     Standard Outputs/.TPearlingYAxis.PlcToNc <-> Inputs/Pearling Y_FromPlc
//   Perlage_Standard/Perlage_Standard Instance <-> NC-Task 1 SAF/Axes/Pearling Z1
//     Standard Inputs/.TPearlingZ1Axis.NcToPlc <-> Outputs/ToPlc
//     Standard Outputs/.TPearlingZ1Axis.PlcToNc <-> Inputs/FromPlc
//   Perlage_Standard/Perlage_Standard Instance <-> NC-Task 1 SAF/Axes/Pearling Z2
//     Standard Inputs/.TPearlingZ2Axis.NcToPlc <-> Outputs/ToPlc
//     Standard Outputs/.TPearlingZ2Axis.PlcToNc <-> Inputs/FromPlc
//   Perlage_Standard/Perlage_Standard Instance <-> NC-Task 1 SAF/Axes/Sharpen
//     Standard Inputs/.TSharpenAxis.NcToPlc <-> Outputs/Sharpen_ToPlc
//     Standard Outputs/.TSharpenAxis.PlcToNc <-> Inputs/Sharpen_FromPlc
//   Perlage_Standard/Perlage_Standard Instance <-> NC-Task 1 SAF/Axes/SharpenEncoder
//     Standard Inputs/.TSharpenEncoder.NcToPlc <-> Outputs/SharpenEncoder_ToPlc
//     Standard Outputs/.TSharpenEncoder.PlcToNc <-> Inputs/SharpenEncoder_FromPlc
//   Perlage_Standard/Perlage_Standard Instance <-> NC-Task 1 SAF/Axes/Table
//     Standard Inputs/.TTableAxis.NcToPlc <-> Outputs/Table_ToPlc
//     Standard Outputs/.TTableAxis.PlcToNc <-> Inputs/Table_FromPlc

CONFIGURATION Perlage_Standard
    RESOURCE PLC ON TwinCAT3
        TASK FastTaskForRS(INTERVAL := T#2ms, PRIORITY := 21);
        TASK Standard(INTERVAL := T#4ms, PRIORITY := 20);
        PROGRAM BG_Serial WITH FastTaskForRS : BG_Serial;
        PROGRAM MAIN WITH Standard : MAIN;
    END_RESOURCE
END_CONFIGURATION

// ---- Data types/TAutoSampling.TcDUT
{attribute 'pack_mode' := '1'}
TYPE TAutoSampling :
STRUCT
	bEnable			: BOOL;
	iPeriod			: INT;
	iBatchSize		: INT;
	iPeriodCnt		: INT;
	iBatchCnt		: INT;
END_STRUCT
END_TYPE

// ---- Data types/TAxisCommands.TcDUT
TYPE TAxisCommands :
	(	AC_None,
		AC_MoveAtSpeed,
		AC_MoveAtRelPos,
		AC_MoveAtAbsPos,
		AC_MoveModulo,
		AC_Stop,
		AC_ForceStop,
		AC_ServoOn,
		AC_ServoOff,
		AC_Init,
		AC_Home,
		AC_MoveHome,
		AC_MoveLimitNeg,
		AC_ClearPosition
	);
END_TYPE

// ---- Data types/TAxisHomingType.TcDUT
TYPE TAxisHomingType :
	(	AHT_NoHoming,
		AHT_OnSensor,
		AHT_OnZeroEncoder
	);
END_TYPE

// ---- Data types/TAxisState.TcDUT
TYPE TAxisState :
	(	AS_PowerOff,
		AS_Powering,
		AS_NotHomed,
		AS_Homing,
		AS_InPosition,
		AS_Moving,
		AS_MovingHoming,
		AS_MovingLimitNeg,
		AS_OnLimitNeg,
		AS_Stopping,
		AS_InError,
		AS_Resetting
	);
END_TYPE

// ---- Data types/TAxisType.TcDUT
TYPE TAxisType :
	(	AT_Standard,
		AT_AX5000
	);
END_TYPE

// ---- Data types/TComIndex.TcDUT
TYPE TComIndex :
	(CI_Pearling:=1);
END_TYPE

// ---- Data types/TConfigFileData.TcDUT
{attribute 'pack_mode' := '1'}
TYPE TConfigFileData :
STRUCT
	bParallelProduction		: BOOL;
	asPearlingData			: ARRAY[PS_SUS..PS_SOUS] OF TPearlingData;
	asStickData				: ARRAY[0..1] OF TStickData;
	sPlateData				: TPlateData;
	sPartData				: TPartDataMMI;
	acVisionRefFileName		: STRING(20);
END_STRUCT
END_TYPE

// ---- Data types/TCounter.TcDUT
{attribute 'pack_mode' := '1'}
TYPE TCounter :
	STRUCT
		sProd							: TprodCounter;
		bResetMTBF						: BOOL;
		dwMeanMTBF					: DWORD;
		adwPearlingMotorRunningHours		: ARRAY[0..1] OF DWORD;
		adwPearlingSpindleRunningHours	: ARRAY[0..1] OF DWORD;
		dwAspirationUseTime				: DWORD;
		dwVacuumUseTime				: DWORD;
		dwMachineOnHours				: DWORD;
		dwInProdHours					: DWORD;
	END_STRUCT
END_TYPE

// ---- Data types/TDashboardCmd.TcDUT
{attribute 'pack_mode' := '1'}
TYPE TDashboardCmd :
STRUCT
		TPearling				: TManButton;
		TLoaderEndOfRecipe		: TManButton;
		TTableTurn				: TManButton;
		TLoaderScanPlateLift1		: TManButton;
		TLoaderScanPlateLift2		: TManButton;
		TLoaderScanPlateReject	: TManButton;
		TPickPlace				: TManButton;
		iScanModel				: INT;
		iMaxScanModel			: INT;
		aiScanPlateOK			: ARRAY[0..2] OF INT;
		aiScanPlateTotal			: ARRAY[0..2] OF INT;
END_STRUCT
END_TYPE

// ---- Data types/TDataLog.TcDUT
{attribute 'pack_mode' := '1'}
TYPE TDataLog :
STRUCT
	bPartReady			: BOOL;
	bEndOfProd			: BOOL;
	sPartStatus			: TPartData;
END_STRUCT
END_TYPE

// ---- Data types/TDynAxisParam.TcDUT
{attribute 'pack_mode' := '1'}
TYPE TDynAxisParam :
STRUCT
	Acc		: LREAL;
	Dec		: LREAL;
	Jerk		: LREAL;
END_STRUCT
END_TYPE

// ---- Data types/TErrors.TcDUT
TYPE TErrors :
(
	ERR_Manager :=0,
	ERR_EmergencyStop,
	ERR_AirPressure,
	ERR_24VPowerSupply,
	ERR_48VPowerSupply,
	ERR_DrivesAreOFF,
	W_LoaderDoorsNotClosed,
	W_PearlingDoorsNotClosed,
	W_NoPowerOnV1,
	W_DoorsNotLocked,
	W_JobPurged,
	ERR_Aspiration,
	ERR_LoaderAxisX,
	ERR_LoaderAxisY,
	ERR_LoaderAxisZ1,
	ERR_LoaderAxisZ2,
	ERR_LoaderAxisTheta,
	ERR_LoaderHead1Vacuum,
	ERR_LoaderHead2Vacuum,
	ERR_LoaderJack,
	ERR_LoaderPlateVacuum,
	ERR_LoaderVision,
	ERR_LoaderNoPartTaken,
	W_LoaderPartsOnPlate,
	ERR_Lift1Drv,
	ERR_Lift2Drv,
	W_LoaderSamplesReady,
	W_RejectChangePlate,
	W_Lift1NeedPlate,
	W_Lift2NeedPlate,
	W_Lift1DrawerNotInPos,
	W_Lift2DrawerNotInPos,
	W_RejectDrawerNotInPos,
	W_RejectPlateNotInPos,
	ERR_BarrelAxis,
	ERR_BarrelJack,
	ERR_BarrelIndex,
	ERR_BarrelStickNotTaken,
	W_BarrelNeedArea1Stick,
	W_BarrelNeedArea2Stick,
	W_BarrelNeedArea3Stick,
	W_BarrelNeedArea4Stick,
	ERR_PearlingAxisX,
	ERR_PearlingAxisY,
	ERR_PearlingAxisZ1,
	ERR_PearlingAxisZ2,
	ERR_PearlingSpindle1,
	ERR_PearlingSpindle2,
	ERR_PearlingGripper1,
	ERR_PearlingGripper2,
	ERR_PearlingMCR,
	ERR_PearlingSecurity,
	ERR_PearlingMotor1,
	ERR_PearlingMotor2,
	ERR_PearlingCurrent1,
	ERR_PearlingCurrent2,
	W_PearlingLeftStickBroken,
	W_PearlingRightStickBroken,
	ERR_TableAxis,
	ERR_TablePearlingAspiration,
	ERR_TableJack,
	ERR_TablePos1Vacuum,
	ERR_TablePos2Vacuum,
	ERR_TablePos3Vacuum,
	ERR_TablePos4Vacuum,
	ERR_TableVacuum4Rotation,
	ERR_BrushAxis,
	ERR_SharpenAxis,
	ERR_SharpenTape,
	ERR_TurnOverAxis,
	ERR_TurnOverJack,
	ERR_TurnOverArmVacuum,
	ERR_TurnOverFixVacuum,
	ERR_VisionNotReady,
	ERR_VisionNotConnected,
	W_VisionInSimulation,
	ERR_Vacuum,
	ERR_BarrelEmpty,
	W_Lift1BadPlate,
	ERR_LoaderZSensorOutOfRange,
	W_PearlingWeight1OutOfTolerance,
	W_PearlingWeight2OutOfTolerance,
	ERR_RejectDrawerOpened,
	W_PearlingLeftSpindleUsed,
	W_PearlingRightSpindleUsed,
	W_PearlingLeftMotorUsed,
	W_PearlingRightMotorUsed,
	ERR_ConfigNotUsable,
	W_PearlingLeftSpindleLimit,
	W_PearlingRightSpindleLimit,
	ERR_Lift1PlateLock,
	ERR_Lift1DrawerLock,
	ERR_Lift2PlateLock,
	ERR_Lift2DrawerLock,
	ERR_TableCleanBrush,
	W_PearlingLeftSpindleHeat,
	W_PearlingRightSpindleHeat
);
END_TYPE

// ---- Data types/TGiver.TcDUT
{attribute 'pack_mode' := '1'}
TYPE TGiver :
	STRUCT
		bHasGiven		: BOOL;		(* Part has been given *)
		bPartDataReady	: BOOL;
		TPartData		: TPartData;
	END_STRUCT
END_TYPE

// ---- Data types/THolderIndex.TcDUT
TYPE THolderIndex :
	(HI_Loader:=0,HI_TableLeftPart1,HI_TableLeftPart2,HI_TableRightPart1,HI_TableRightPart2,HI_TurnOver,HI_Unloader,HI_END);
END_TYPE

// ---- Data types/TLiftPos.TcDUT
TYPE TLiftPos :
	(
		LP_OnPlate := 0,
		LP_OnPlateLoad,
		LP_Moving,
		LP_Empty,
		LP_Full,
		LP_OpenDrawer
	);
END_TYPE

// ---- Data types/TLiftType.TcDUT
TYPE TLiftType :
	(LT_LOADER := 0,LT_UNLOADER, LT_REJECT);
END_TYPE

// ---- Data types/TLoaderAxis.TcDUT
TYPE TLoaderAxis :
	(
		LA_X := 0,
		LA_Y,
		LA_Z1,
		LA_Z2,
		LA_THETA
	);
END_TYPE

// ---- Data types/TLoaderDropMode.TcDUT
TYPE TLoaderDropMode :
	(
		LDM_DropAndGoUp := 0,
		LDM_DropAndWaitDown,
		LDM_WaitDownAndDrop
	);
END_TYPE

// ---- Data types/TLoaderHead.TcDUT
TYPE TLoaderHead :
	(
		LH_Head1 := 0,
		LH_Head2
	);
END_TYPE

// ---- Data types/TLoaderModulePos.TcDUT
TYPE TLoaderModulePos :
	(
			LMP_Reject :=0,
			LMP_Lift1,
			LMP_Lift2,
			LMP_Table,
			LMP_TurnOverFix,
			LMP_TurnOverArm,
			LMP_Sample
	);
END_TYPE

// ---- Data types/TLoaderPlatePos.TcDUT
TYPE TLoaderPlatePos :
	(
		LPP_Reject := 0,
		LPP_Lift1,
		LPP_Lift2
	);
END_TYPE

// ---- Data types/TLoaderSynchro.TcDUT
TYPE TLoaderSynchro :
	(LS_TableLeftPart1 := 0,LS_TableLeftPart2,LS_TableRightPart1,LS_TableRightPart2,LS_END);
END_TYPE

// ---- Data types/TLoaderTakeMode.TcDUT
TYPE TLoaderTakeMode :
	(
		LTM_GoDownAndVacuum := 0,
		LTM_VacuumAndGoDown
	);
END_TYPE

// ---- Data types/TLoaderTeachedAxis.TcDUT
TYPE TLoaderTeachedAxis :
	(
		LTA_X := 0,
		LTA_Y,
		LTA_Z,
		LTA_THETA
	);
END_TYPE

// ---- Data types/TLoaderTeachOffset.TcDUT
TYPE TLoaderTeachOffset :
	(
			LTO_Z1			:=0,
			LTO_Z2,
			LTO_Plate,
			LTO_Vision,
			LTO_ZSensor,
			LTO_END
	);
END_TYPE

// ---- Data types/TLoaderTeachPos.TcDUT
TYPE TLoaderTeachPos :
	(
			LTP_Reject :=0,
			LTP_Lift1,
			LTP_Lift2,
			LTP_TableSideALayering1,
			LTP_TableSideBLayering1,
			LTP_CleanBrush,
			LTP_TurnOverFix,
			LTP_TurnOverArm,
			LTP_TableSideALayering2,
			LTP_TableSideBLayering2,
			LTP_BulkBox,
			LTP_RejectBulkBox,
			LTP_END
	);
END_TYPE

// ---- Data types/TMachineData.TcDUT
{attribute 'pack_mode' := '1'}
TYPE TMachineData :
STRUCT
	bReadyForChangeJob		: BOOL;
	bMachineInitDone			: BOOL;
	bResetErrors				: BOOL;
	bClearRates				: BOOL;
	bNewJob				: BOOL;
	bCloseJob				: BOOL;
	bPurgeJob				: BOOL;
	bMondemaMode			: BOOL;
	abErrorsTable			: ARRAY[0..C_MAX_NB_OF_ERRORS] OF BOOL;
	abValErrorsTable			: ARRAY[0..C_MAX_NB_OF_ERRORS] OF BOOL;
	eCurrentMode			: TMachineMode := MM_Stopped;
	acPartName				: STRING(8);
	iMajorVersion				: INT;
	iMinorVersion				: INT;
	sModeMask				: TMachineModeMask;
	sModeReq				: TMachineModeMask;
	sModLoader				: TModuleData;
	sModTable				: TModuleData;
	sModPearling			: TModuleData;
	sModSharpen			: TModuleData;
	sModTurnOver			: TModuleData;
	sModBarrel				: TModuleData;
	sModLift1				: TModuleData;
	sModLift2				: TModuleData;
	sModReject				: TModuleData;
	sModVision				: TModuleData;
	sModUtilities				: TModuleData;
	sMachineOpt				: TMachineOptions;
	sProdData				: TProductionlot;
	sProdStats				: TProductionStats;
	sPartDataForLog			: TDataLog;
	sMachineManualCmd		: TMachineManual;
	sOperatorReq			: TOperatorReq;
	asStickData				: ARRAY[0..1] OF TStickDataMMI;
	asPearlsData				: ARRAY[0..1] OF TMMIPearlData;
	sStickDataShared			: TStickDataMMIShared;
	bEmergencyStop			: BOOL;
	bDoorsPearling			: BOOL;
	bDoorsLoader			: BOOL;
	bSavePersistent			: BOOL;
	eManagerRunStep		: TModuleSteps;
	sDashboardCmd			: TDashboardCmd;
	bSimPearling				: BOOL;
	asProbingLog			: ARRAY[0..1] OF  TProbingLog;
	sProductionCmd			: TProductionCmd;
	dwStartJobElapsedTime	: DWORD;
	sCounter					: TCounter;
END_STRUCT
END_TYPE

// ---- Data types/TMachineManual.TcDUT
{attribute 'pack_mode' := '1'}
TYPE TMachineManual :
STRUCT
	bCanLockDoor		: BOOL;
	bLockDoor			: BOOL;
	bCanUnlockDoor		: BOOL;
	bUnlockDoor			: BOOL;
END_STRUCT
END_TYPE

// ---- Data types/TMachineMode.TcDUT
TYPE TMachineMode :
	(	MM_Stopped:=0,
		MM_Init,
		MM_Ready,
		MM_Running,
		MM_Dashboard,
		MM_Stopping,
		MM_Manual,
		MM_Pause,
		MM_Pausing,
		MM_ForceStop,
		MM_Purging
	);
END_TYPE

// ---- Data types/TMachineModeMask.TcDUT
{attribute 'pack_mode' := '1'}
TYPE TMachineModeMask :
STRUCT
	bStop			: BOOL;
	bInit				: BOOL;
	bRun			: BOOL;
	bManual			: BOOL;
	bPurge			: BOOL;
	bPause			: BOOL;
	bDashboard		: BOOL;
END_STRUCT
END_TYPE

// ---- Data types/TMachineOptions.TcDUT
{attribute 'pack_mode' := '1'}
TYPE TMachineOptions :
STRUCT
	TurnOver		: BOOL;
	RTPearling		: BOOL;
	AutoSampling	: BOOL;
	bDisableCleanAfterPearling		: BOOL;
	bDisableVision	: BOOL;
	bSpeedModeSlow	: BOOL;
END_STRUCT
END_TYPE

// ---- Data types/TMachineSafety.TcDUT
{attribute 'pack_mode' := '1'}
TYPE TMachineSafety :
STRUCT
	bCanLockDoor		: BOOL;
	bLockDoor			: BOOL;
	bCanUnlockDoor		: BOOL;
	bUnlockDoor			: BOOL;
END_STRUCT
END_TYPE

// ---- Data types/TManagerPartStatus.TcDUT
TYPE TManagerPartStatus :
	(
		MPS_NoPart,
		MPS_NeedPearling,
		MPS_ReadyToMove,
		MPS_PartBusy
	);
END_TYPE

// ---- Data types/TManBarrel.TcDUT
{attribute 'pack_mode' := '1'}
TYPE TManBarrel :
	STRUCT
		iIndexSection				: INT;
		iIndexPosition 			: INT;
		iPosition					: INT;
		bStickPresent 			: BOOL;
		TBarrelAxis				: TManDrive;
		TBarrelAxisTakenPos		: TManDrivePos;
		TBarrelAxisCheckPos		: TManDrivePos;
		TMoveJackUp			: TManButton;
		TIndexTable				: TManButton;
		TMoveTaken				: TManBarrelAxisPosition;
		TMoveCheck				: TManBarrelAxisPosition;
	END_STRUCT
END_TYPE

// ---- Data types/TManBarrelAxisPosition.TcDUT
{attribute 'pack_mode' := '1'}
TYPE TManBarrelAxisPosition :
STRUCT
		TMove1Step				: TManButton;
		TMoveSectionA			: TManButton;
		TMoveSectionB			: TManButton;
		TMoveSectionC			: TManButton;
		TMoveSectionD			: TManButton;
END_STRUCT
END_TYPE

// ---- Data types/TManButton.TcDUT
{attribute 'pack_mode' := '1'}
TYPE TManButton :
	STRUCT
		Activate		: BOOL	 := FALSE;
		Enable		: BOOL	 := FALSE;
	END_STRUCT
END_TYPE

// ---- Data types/TManDrive.TcDUT
{attribute 'pack_mode' := '1'}
TYPE TManDrive :
	STRUCT
		CurrentPos		: LREAL;
		JogStep			: LREAL;
		Specific			: TManButton;
		ServoON		: TManButton;
		Home			: TManButton;
		MoveFw			: TManButton;
		MoveBw			: TManButton;
		UseHours		: DWORD;
		ResetUseTime	: TManButton;
	END_STRUCT
END_TYPE

// ---- Data types/TManDrivePos.TcDUT
{attribute 'pack_mode' := '1'}
TYPE TManDrivePos :
	STRUCT
		Teach			: BOOL	 := FALSE;
		TeachedPos		: LREAL;
		MoveToTeach	: TManButton;
	END_STRUCT
END_TYPE

// ---- Data types/TManLift.TcDUT
{attribute 'pack_mode' := '1'}
TYPE TManLift :
	STRUCT
		TLiftAxis				: TManDrive;
		TLiftAxisFullPos		: TManDrivePos;
		TLiftAxisEmptyPos		: TManDrivePos;
		TLiftAxisLoadPos		: TManDrivePos;
		TLiftAxisZOffset		: TManDrivePos;
		TMoveToPlate			: TManButton;
		TMoveToPlateVision		: TManButton;
		bDrawerInPos 			: BOOL;
		bPlateInPos 			: BOOL;
		lrPlatePos				: LREAL;
		TLockDrawer				: TManButton;
		TLockPlate				: TManButton;
	END_STRUCT
END_TYPE

// ---- Data types/TManLoader.TcDUT
{attribute 'pack_mode' := '1'}
TYPE TManLoader :
	STRUCT
		eTableSide				: TTableSide;
		bAxisZSafe				: ARRAY[0..1] OF BOOL;
		aTAxis					: ARRAY[0..4] OF TManDrive;
		aTAxisPos				: ARRAY[0..4] OF TManDrivePos;
		TSafe					: TManButton;
		TVisionCalibration		: TManButton;
		THead1Vacuum			: TManButton;
		THead2Vacuum			: TManButton;
		TPlateVacuum			: TManButton;
		alrVaccumValue			: ARRAY[0..1] OF  LREAL;
		alrVaccumThershold		: ARRAY[0..1] OF  LREAL;
		TMovePlateTakerDown		: TManButton;
		TAspirationBrush		: TManButton;
		lrSensorAdjust			: LREAL;
		lrSensorMeasure			: LREAL;
		wRobotPos				: WORD;
		TZSensorTeach			: TManButton;
		TMoveVision2Table		: TManButton;
		TMoveVision2Lift		: TManButton;
		wMoveVision2LiftPos		: WORD;
	END_STRUCT
END_TYPE

// ---- Data types/TManPearling.TcDUT
{attribute 'pack_mode' := '1'}
TYPE TManPearling :
STRUCT
	e_TeachPos					: TPearlingTeachPos;
	eTableSide					: TTableSide;
	bAxisZSafe					: ARRAY[0..1] OF BOOL;
	aiMotorSpeed				: ARRAY[0..1] OF INT;
	arMotorCurrent				: ARRAY[0..1] OF REAL;
	adwMotorRunningHours		: ARRAY[0..1] OF DWORD;
	adwSpindleRunningHours		: ARRAY[0..1] OF DWORD;
	aTAxis						: ARRAY[0..3] OF TManDrive;
	aTAxisPos					: ARRAY[0..3] OF TManDrivePos;
	aTStartMotor				: ARRAY[0..1] OF TManButton;
	aTOpenChuck					: ARRAY[0..1] OF TManButton;
	aTEjectStick				: ARRAY[0..1] OF TManButton;
	aTActivateBlowing			: ARRAY[0..1] OF TManButton;
	TSafe						: TManButton;
	aTCalibrateWeight			: ARRAY[0..1] OF TManButton;
	TResetMotorUseTime			: ARRAY[0..1] OF TManButton;
	TResetSpindleUseTime		: ARRAY[0..1] OF TManButton;
	lrWeightStepOnZ				: LREAL;
	alrWeightTableLeft			: ARRAY[0..C_WEIGHT_TABLE_MAX] OF LREAL;
	alrWeightTableRight			: ARRAY[0..C_WEIGHT_TABLE_MAX] OF LREAL;
	bWeightTableLeftValid		: BOOL;
	bWeightTableRightValid		: BOOL;
	TActivateAspirationTable	: ARRAY[0..1] OF TManButton;
	TActivateAspirationSharpen	: TManButton;
	aiSpindleSpeedSetpoint		: ARRAY[0..1] OF INT;
	iCurrentMotorMinTh			: INT;
	iCurrentMotorWarnTh			: INT;
	iCurrentMotorMaxTh			: INT;
	aiMotorStartedTimeout		: ARRAY[0..1] OF INT;
	aiMotorStoppedTimeout		: ARRAY[0..1] OF INT;
	alrRatiog2mm				: ARRAY[0..1] OF LREAL;
	aiDistanceSensor			: ARRAY[0..1] OF INT;
	iWeightSensor				: INT;
	adwPearlsCounter			: ARRAY[0..1] OF DWORD;
END_STRUCT
END_TYPE

// ---- Data types/TManReject.TcDUT
{attribute 'pack_mode' := '1'}
TYPE TManReject :
	STRUCT
		bDrawerInPos 			: BOOL;
		bPlateInPos 				: BOOL;
	END_STRUCT
END_TYPE

// ---- Data types/TManSharpen.TcDUT
{attribute 'pack_mode' := '1'}
TYPE TManSharpen :
STRUCT
	TSharpenAxis				: TManDrive;
	TMove2NextTapePos			: TManButton;
	bTapeNotEmpty				: BOOL;
	lrStep						: LREAL;
END_STRUCT
END_TYPE

// ---- Data types/TManTable.TcDUT
{attribute 'pack_mode' := '1'}
TYPE TManTable :
STRUCT
	TAxisTable						: TManDrive;
	TAxisTableLoading12Pos			: TManDrivePos;
	TAxisTableLoading34Pos			: TManDrivePos;
	TAxisBrush						: TManDrive;
	aTAxisBrushParkPos				:  ARRAY[0..1] OF  TManDrivePos;
	aTAxisBrushWorkPos				:  ARRAY[0..1] OF  TManDrivePos;
	TAspirationDown					: TManButton;
	TIndexTable						: TManButton;
	TPlate1Vacuum					: TManButton;
	TPlate2Vacuum					: TManButton;
	TPlate3Vacuum					: TManButton;
	TPlate4Vacuum					: TManButton;
	alrVaccumValue					: ARRAY[0..3] OF  LREAL;
	alrVaccumThershold				: ARRAY[0..3] OF  LREAL;
	TAspirationBrush				: TManButton;
	TCleanBrushDown					: TManButton;
END_STRUCT
END_TYPE

// ---- Data types/TManTurnOver.TcDUT
{attribute 'pack_mode' := '1'}
TYPE TManTurnOver :
STRUCT
	TTurnOverAxis				: TManDrive;
	TTurnOverAxisIndexPos		: TManDrivePos;
	TTurnOverAxisFlippedPos		: TManDrivePos;
	TJack						: TManButton;
	TActivateArmVacuum			: TManButton;
	TActivateFixVacuum			: TManButton;
	TActivateCleaningBlow			: TManButton;
END_STRUCT
END_TYPE

// ---- Data types/TManualData.TcDUT
{attribute 'pack_mode' := '1'}
TYPE TManualData :
STRUCT
	TLoaderManual				: TManLoader;
	TTableManual				: TManTable;
	TPearlingManual				: TManPearling;
	TSharpenManual				: TManSharpen;
	TTurnOverManual				: TManTurnOver;
	TBarrelManual				: TManBarrel;
	TLift1Manual					: TManLift;
	TLift2Manual					: TManLift;
	TRejectManual				: TManReject;
	TVisionManual				: TManVision;
	TUtilitiesManual				: TManUtilities;
	sVacuumSettingsMMI			: TVacuumSettingsMMI;
END_STRUCT
END_TYPE

// ---- Data types/TManUtilities.TcDUT
{attribute 'pack_mode' := '1'}
TYPE TManUtilities :
	STRUCT
		TAspiration				: TManButton;
		TVacuum				: TManButton;
		bPowerIsOn				: BOOL;
		bDrivesIsOn				: BOOL;
		b24VOK					: BOOL;
		b48VOK					: BOOL;
		bAirPressureOK			: BOOL;
		bMainVacuumOK			: BOOL;
		bAspirationOK			: BOOL;
		bAspirationIsOn			: BOOL;
		TResetAspirationUseTime	: TManButton;
		dwAspirationUseTime		: DWORD;
		TResetVacuumUseTime	: TManButton;
		dwVacuumUseTime		: DWORD;
	END_STRUCT
END_TYPE

// ---- Data types/TManVision.TcDUT
{attribute 'pack_mode' := '1'}
TYPE TManVision :
	STRUCT
		TInit					: TManButton;
		TAnalyse			: TManButton;
		TRun				: TManButton;
		TInitTime			: TIMESTRUCT;
		TAnalyseTime		: TIMESTRUCT;
		acVisionRecipeName	: STRING(20);
		bConnected			: BOOL;
		bReady				: BOOL;
		bSimRecipe			: BOOL;
		iUseModel			: INT;
		iMaxModel			: INT;
		TPartData			: TVisionPartData;
		bPartDataValid		: BOOL;
		bConfigMode			: TManButton ;
	END_STRUCT
END_TYPE

// ---- Data types/TMCRCommands.TcDUT
TYPE TMCRCommands :
	(	MCRC_None,
		MCRC_ConfigMeasure,
		MCRC_SetRatio,
		MCRC_StartPower,
		MCRC_ReadCurrent,
		MCRC_UpdateMemory,
		MCRC_DefineCurrentThr,
		MCRC_GetPower,
		MCRC_GetParam,
		MCRC_ReadSpeed,
		MCRC_SetSpeed,
		MCRC_GetVersion,
		MCRC_SetParam,
		MCRC_DefineMachineID,
		MCRC_GetStatus
	);
END_TYPE

// ---- Data types/TMDE.TcDUT
{attribute 'pack_mode' := '1'}
TYPE TMDE :
STRUCT
	dwPceBad		: DWORD;
	dwPceGood		: DWORD;
	iPertCode		: INT;
	iStatus			: INT;
END_STRUCT
END_TYPE

// ---- Data types/TMDEStatus.TcDUT
TYPE TMDEStatus :
	(	MDE_Alarm,
		MDE_Production,
		MDE_Standby,
		MDE_Maintenance	);
END_TYPE

// ---- Data types/TMMIPearlData.TcDUT
{attribute 'pack_mode' := '1'}
TYPE TMMIPearlData :
STRUCT
	bNewPearl			: BOOL;
	bNewPart			: BOOL;
	iPearlNb				: INT;
	iRate				: INT;
	bPearlingTop			: BOOL;
	lrPearlingCalcPos		: LREAL;
	lrPearlingMeasurePos	: LREAL;
	lrDeltaCurrent			: LREAL;
	lrCorrectionMCR		: LREAL;
	lrDispersion			: LREAL;
	lrSensorProbePos		: LREAL;
	lrSensorPearlPos		: LREAL;
	lrDeltaWeight			: LREAL;
	iVacuumFlow				: INT;
END_STRUCT
END_TYPE

// ---- Data types/TModuleCommands.TcDUT
TYPE TModuleCommands :
	(
		MC_NoCmd,
		MC_Init,
		MC_Manual,
		MC_Stop,
		MC_Run
	);
END_TYPE

// ---- Data types/TModuleData.TcDUT
{attribute 'pack_mode' := '1'}
TYPE TModuleData :
STRUCT
	bInitDone	: BOOL			:= FALSE;
	bRunning	: BOOL			:= FALSE;
	bInError		: BOOL			:= FALSE;
	bInterlocked	: BOOL			:= FALSE;
	bWarning	: BOOL			:= FALSE;
	bStepMode	: BOOL			:= FALSE;
	bWaitStep	: BOOL			:= FALSE;
	eStatus 		: TModuleStatus	 := MS_Stopped;
	eStep		: TModuleSteps	:= SP_InitStp1;
END_STRUCT
END_TYPE

// ---- Data types/TModuleStatus.TcDUT
TYPE TModuleStatus :
	(	MS_Stopped:=0,
		MS_Init,
		MS_Running,
		MS_Ready,
		MS_Manual,
		MS_Paused
	);
END_TYPE

// ---- Data types/TModuleSteps.TcDUT
TYPE TModuleSteps :
(
	SP_InitStp0:=0,SP_InitStp1,SP_InitStp2,SP_InitStp3,SP_InitStp4,SP_InitStp5,SP_InitStp6,SP_InitStp7,SP_InitStp8,SP_InitStp9,
	SP_InitStp10:=10,SP_InitStp11,SP_InitStp12,SP_InitStp13,SP_InitStp14,SP_InitStp15,SP_InitStp16,SP_InitStp17,SP_InitStp18,SP_InitStp19,
	SP_InitStp20:=20,SP_InitStp21,SP_InitStp22,SP_InitStp23,SP_InitStp24,SP_InitStp25,SP_InitStp26,SP_InitStp27,SP_InitStp28,SP_InitStp29,
	SP_InitStp30:=30,SP_InitStp31,SP_InitStp32,SP_InitStp33,SP_InitStp34,SP_InitStp35,SP_InitStp36,SP_InitStp37,SP_InitStp38,SP_InitStp39,
	SP_InitStp40:=40,SP_InitStp41,SP_InitStp42,SP_InitStp43,SP_InitStp44,SP_InitStp45,SP_InitStp46,SP_InitStp47,SP_InitStp48,SP_InitStp49,
	SP_InitStp50:=50,SP_InitStp51,SP_InitStp52,SP_InitStp53,SP_InitStp54,SP_InitStp55,SP_InitStp56,SP_InitStp57,SP_InitStp58,SP_InitStp59,
	SP_InitStp90:=90,SP_InitStp91,SP_InitStp92,SP_InitStp93,SP_InitStp94,SP_InitStp95,SP_InitStp96,SP_InitStp97,SP_InitStp98,SP_InitStp99,
	SP_RunStp0:=1000,SP_RunStp1,SP_RunStp2,SP_RunStp3,SP_RunStp4,SP_RunStp5,SP_RunStp6,SP_RunStp7,SP_RunStp8,SP_RunStp9,
	SP_RunStp10:=1010,SP_RunStp11,SP_RunStp12,SP_RunStp13,SP_RunStp14,SP_RunStp15,SP_RunStp16,SP_RunStp17,SP_RunStp18,SP_RunStp19,
	SP_RunStp20:=1020,SP_RunStp21,SP_RunStp22,SP_RunStp23,SP_RunStp24,SP_RunStp25,SP_RunStp26,SP_RunStp27,SP_RunStp28,SP_RunStp29,
	SP_RunStp30:=1030,SP_RunStp31,SP_RunStp32,SP_RunStp33,SP_RunStp34,SP_RunStp35,SP_RunStp36,SP_RunStp37,SP_RunStp38,SP_RunStp39,
	SP_RunStp40:=1040,SP_RunStp41,SP_RunStp42,SP_RunStp43,SP_RunStp44,SP_RunStp45,SP_RunStp46,SP_RunStp47,SP_RunStp48,SP_RunStp49,
	SP_RunStp50:=1050,SP_RunStp51,SP_RunStp52,SP_RunStp53,SP_RunStp54,SP_RunStp55,SP_RunStp56,SP_RunStp57,SP_RunStp58,SP_RunStp59,
	SP_RunStp60:=1060,SP_RunStp61,SP_RunStp62,SP_RunStp63,SP_RunStp64,SP_RunStp65,SP_RunStp66,SP_RunStp67,SP_RunStp68,SP_RunStp69,
	SP_RunStp70:=1070,SP_RunStp71,SP_RunStp72,SP_RunStp73,SP_RunStp74,SP_RunStp75,SP_RunStp76,SP_RunStp77,SP_RunStp78,SP_RunStp79,
	SP_RunStp80:=1080,SP_RunStp81,SP_RunStp82,SP_RunStp83,SP_RunStp84,SP_RunStp85,SP_RunStp86,SP_RunStp87,SP_RunStp88,SP_RunStp89,
	SP_RunStp90:=1090,SP_RunStp91,SP_RunStp92,SP_RunStp93,SP_RunStp94,SP_RunStp95,SP_RunStp96,SP_RunStp97,SP_RunStp98,SP_RunStp99,
	SP_RunStp100:=1100,SP_RunStp101,SP_RunStp102,SP_RunStp103,SP_RunStp104,SP_RunStp105,SP_RunStp106,SP_RunStp107,SP_RunStp108,SP_RunStp109,
	SP_RunStp110:=1110,SP_RunStp111,SP_RunStp112,SP_RunStp113,SP_RunStp114,SP_RunStp115,SP_RunStp116,SP_RunStp117,SP_RunStp118,SP_RunStp119,
	SP_RunStp120:=1120,SP_RunStp121,SP_RunStp122,SP_RunStp123,SP_RunStp124,SP_RunStp125,SP_RunStp126,SP_RunStp127,SP_RunStp128,SP_RunStp129,
	SP_RunStp130:=1130,SP_RunStp131,SP_RunStp132,SP_RunStp133,SP_RunStp134,SP_RunStp135,SP_RunStp136,SP_RunStp137,SP_RunStp138,SP_RunStp139,
	SP_RunStp140:=1140,SP_RunStp141,SP_RunStp142,SP_RunStp143,SP_RunStp144,SP_RunStp145,SP_RunStp146,SP_RunStp147,SP_RunStp148,SP_RunStp149,
	SP_RunStp150:=1150,SP_RunStp151,SP_RunStp152,SP_RunStp153,SP_RunStp154,SP_RunStp155,SP_RunStp156,SP_RunStp157,SP_RunStp158,SP_RunStp159,
	SP_RunStp160:=1160,SP_RunStp161,SP_RunStp162,SP_RunStp163,SP_RunStp164,SP_RunStp165,SP_RunStp166,SP_RunStp167,SP_RunStp168,SP_RunStp169,
	SP_RunStp170:=1170,SP_RunStp171,SP_RunStp172,SP_RunStp173,SP_RunStp174,SP_RunStp175,SP_RunStp176,SP_RunStp177,SP_RunStp178,SP_RunStp179,
	SP_RunStp180:=1180,SP_RunStp181,SP_RunStp182,SP_RunStp183,SP_RunStp184,SP_RunStp185,SP_RunStp186,SP_RunStp187,SP_RunStp188,SP_RunStp189,
	SP_RunStp190:=1190,SP_RunStp191,SP_RunStp192,SP_RunStp193,SP_RunStp194,SP_RunStp195,SP_RunStp196,SP_RunStp197,SP_RunStp198,SP_RunStp199,
	SP_RunStp200:=1200,SP_RunStp201,SP_RunStp202,SP_RunStp203,SP_RunStp204,SP_RunStp205,SP_RunStp206,SP_RunStp207,SP_RunStp208,SP_RunStp209,
	SP_RunStp210:=1210,SP_RunStp211,SP_RunStp212,SP_RunStp213,SP_RunStp214,SP_RunStp215,SP_RunStp216,SP_RunStp217,SP_RunStp218,SP_RunStp219,
	SP_RunStp220:=1220,SP_RunStp221,SP_RunStp222,SP_RunStp223,SP_RunStp224,SP_RunStp225,SP_RunStp226,SP_RunStp227,SP_RunStp228,SP_RunStp229,
	SP_RunStp230:=1230,SP_RunStp231,SP_RunStp232,SP_RunStp233,SP_RunStp234,SP_RunStp235,SP_RunStp236,SP_RunStp237,SP_RunStp238,SP_RunStp239,
	SP_RunStp240:=1240,SP_RunStp241,SP_RunStp242,SP_RunStp243,SP_RunStp244,SP_RunStp245,SP_RunStp246,SP_RunStp247,SP_RunStp248,SP_RunStp249,
	SP_RunStp250:=1250,SP_RunStp251,SP_RunStp252,SP_RunStp253,SP_RunStp254,SP_RunStp255,SP_RunStp256,SP_RunStp257,SP_RunStp258,SP_RunStp259,
	SP_RunStp260:=1260,SP_RunStp261,SP_RunStp262,SP_RunStp263,SP_RunStp264,SP_RunStp265,SP_RunStp266,SP_RunStp267,SP_RunStp268,SP_RunStp269,
	SP_RunStp270:=1270,SP_RunStp271,SP_RunStp272,SP_RunStp273,SP_RunStp274,SP_RunStp275,SP_RunStp276,SP_RunStp277,SP_RunStp278,SP_RunStp279,
	SP_RunStp280:=1280,SP_RunStp281,SP_RunStp282,SP_RunStp283,SP_RunStp284,SP_RunStp285,SP_RunStp286,SP_RunStp287,SP_RunStp288,SP_RunStp289,
	SP_RunStp290:=1290,SP_RunStp291,SP_RunStp292,SP_RunStp293,SP_RunStp294,SP_RunStp295,SP_RunStp296,SP_RunStp297,SP_RunStp298,SP_RunStp299,
	SP_RunStp300:=1300,SP_RunStp301,SP_RunStp302,SP_RunStp303,SP_RunStp304,SP_RunStp305,SP_RunStp306,SP_RunStp307,SP_RunStp308,SP_RunStp309,
	SP_RunStp310:=1310,SP_RunStp311,SP_RunStp312,SP_RunStp313,SP_RunStp314,SP_RunStp315,SP_RunStp316,SP_RunStp317,SP_RunStp318,SP_RunStp319,
	SP_RunStp320:=1320,SP_RunStp321,SP_RunStp322,SP_RunStp323,SP_RunStp324,SP_RunStp325,SP_RunStp326,SP_RunStp327,SP_RunStp328,SP_RunStp329,
	SP_RunStp330:=1330,SP_RunStp331,SP_RunStp332,SP_RunStp333,SP_RunStp334,SP_RunStp335,SP_RunStp336,SP_RunStp337,SP_RunStp338,SP_RunStp339,
	SP_RunStp340:=1340,SP_RunStp341,SP_RunStp342,SP_RunStp343,SP_RunStp344,SP_RunStp345,SP_RunStp346,SP_RunStp347,SP_RunStp348,SP_RunStp349,
	SP_RunStp350:=1350,SP_RunStp351,SP_RunStp352,SP_RunStp353,SP_RunStp354,SP_RunStp355,SP_RunStp356,SP_RunStp357,SP_RunStp358,SP_RunStp359,
	SP_RunStp360:=1360,SP_RunStp361,SP_RunStp362,SP_RunStp363,SP_RunStp364,SP_RunStp365,SP_RunStp366,SP_RunStp367,SP_RunStp368,SP_RunStp369,
	SP_RunStp370:=1370,SP_RunStp371,SP_RunStp372,SP_RunStp373,SP_RunStp374,SP_RunStp375,SP_RunStp376,SP_RunStp377,SP_RunStp378,SP_RunStp379,
	SP_RunStp380:=1380,SP_RunStp381,SP_RunStp382,SP_RunStp383,SP_RunStp384,SP_RunStp385,SP_RunStp386,SP_RunStp387,SP_RunStp388,SP_RunStp389,
	SP_RunStp390:=1390,SP_RunStp391,SP_RunStp392,SP_RunStp393,SP_RunStp394,SP_RunStp395,SP_RunStp396,SP_RunStp397,SP_RunStp398,SP_RunStp399,
	SP_RunStp400:=1400,SP_RunStp401,SP_RunStp402,SP_RunStp403,SP_RunStp404,SP_RunStp405,SP_RunStp406,SP_RunStp407,SP_RunStp408,SP_RunStp409,
	SP_RunStp410:=1410,SP_RunStp411,SP_RunStp412,SP_RunStp413,SP_RunStp414,SP_RunStp415,SP_RunStp416,SP_RunStp417,SP_RunStp418,SP_RunStp419,
	SP_RunStp420:=1420,SP_RunStp421,SP_RunStp422,SP_RunStp423,SP_RunStp424,SP_RunStp425,SP_RunStp426,SP_RunStp427,SP_RunStp428,SP_RunStp429,
	SP_RunStp430:=1430,SP_RunStp431,SP_RunStp432,SP_RunStp433,SP_RunStp434,SP_RunStp435,SP_RunStp436,SP_RunStp437,SP_RunStp438,SP_RunStp439,
	SP_RunStp440:=1440,SP_RunStp441,SP_RunStp442,SP_RunStp443,SP_RunStp444,SP_RunStp445,SP_RunStp446,SP_RunStp447,SP_RunStp448,SP_RunStp449,
	SP_RunStp450:=1450,SP_RunStp451,SP_RunStp452,SP_RunStp453,SP_RunStp454,SP_RunStp455,SP_RunStp456,SP_RunStp457,SP_RunStp458,SP_RunStp459,
	SP_RunStp460:=1460,SP_RunStp461,SP_RunStp462,SP_RunStp463,SP_RunStp464,SP_RunStp465,SP_RunStp466,SP_RunStp467,SP_RunStp468,SP_RunStp469,
	SP_RunStp470:=1470,SP_RunStp471,SP_RunStp472,SP_RunStp473,SP_RunStp474,SP_RunStp475,SP_RunStp476,SP_RunStp477,SP_RunStp478,SP_RunStp479,
	SP_RunStp480:=1480,SP_RunStp481,SP_RunStp482,SP_RunStp483,SP_RunStp484,SP_RunStp485,SP_RunStp486,SP_RunStp487,SP_RunStp488,SP_RunStp489,
	SP_RunStp490:=1490,SP_RunStp491,SP_RunStp492,SP_RunStp493,SP_RunStp494,SP_RunStp495,SP_RunStp496,SP_RunStp497,SP_RunStp498,SP_RunStp499,
	SP_RunStp500:=1500,SP_RunStp501,SP_RunStp502,SP_RunStp503,SP_RunStp504,SP_RunStp505,SP_RunStp506,SP_RunStp507,SP_RunStp508,SP_RunStp509,
	SP_RunStp510:=1510,SP_RunStp511,SP_RunStp512,SP_RunStp513,SP_RunStp514,SP_RunStp515,SP_RunStp516,SP_RunStp517,SP_RunStp518,SP_RunStp519,
	SP_RunStp520:=1520,SP_RunStp521,SP_RunStp522,SP_RunStp523,SP_RunStp524,SP_RunStp525,SP_RunStp526,SP_RunStp527,SP_RunStp528,SP_RunStp529,
	SP_RunStp530:=1530,SP_RunStp531,SP_RunStp532,SP_RunStp533,SP_RunStp534,SP_RunStp535,SP_RunStp536,SP_RunStp537,SP_RunStp538,SP_RunStp539,
	SP_RunStp540:=1540,SP_RunStp541,SP_RunStp542,SP_RunStp543,SP_RunStp544,SP_RunStp545,SP_RunStp546,SP_RunStp547,SP_RunStp548,SP_RunStp549,
	SP_RunStp550:=1550,SP_RunStp551,SP_RunStp552,SP_RunStp553,SP_RunStp554,SP_RunStp555,SP_RunStp556,SP_RunStp557,SP_RunStp558,SP_RunStp559,
	SP_RunStp560:=1560,SP_RunStp561,SP_RunStp562,SP_RunStp563,SP_RunStp564,SP_RunStp565,SP_RunStp566,SP_RunStp567,SP_RunStp568,SP_RunStp569,
	SP_RunStp570:=1570,SP_RunStp571,SP_RunStp572,SP_RunStp573,SP_RunStp574,SP_RunStp575,SP_RunStp576,SP_RunStp577,SP_RunStp578,SP_RunStp579,
	SP_RunStp580:=1580,SP_RunStp581,SP_RunStp582,SP_RunStp583,SP_RunStp584,SP_RunStp585,SP_RunStp586,SP_RunStp587,SP_RunStp588,SP_RunStp589,
	SP_RunStp590:=1590,SP_RunStp591,SP_RunStp592,SP_RunStp593,SP_RunStp594,SP_RunStp595,SP_RunStp596,SP_RunStp597,SP_RunStp598,SP_RunStp599,
	SP_ManualStp0:=2000,SP_ManualStp1,SP_ManualStp2,SP_ManualStp3,SP_ManualStp4,SP_ManualStp5,SP_ManualStp6,SP_ManualStp7,SP_ManualStp8,SP_ManualStp9,
	SP_ManualStp10:=2010,SP_ManualStp11,SP_ManualStp12,SP_ManualStp13,SP_ManualStp14,SP_ManualStp15,SP_ManualStp16,SP_ManualStp17,SP_ManualStp18,SP_ManualStp19,
	SP_ManualStp20:=2020,SP_ManualStp21,SP_ManualStp22,SP_ManualStp23,SP_ManualStp24,SP_ManualStp25,SP_ManualStp26,SP_ManualStp27,SP_ManualStp28,SP_ManualStp29,
	SP_ManualStp30:=2030,SP_ManualStp31,SP_ManualStp32,SP_ManualStp33,SP_ManualStp34,SP_ManualStp35,SP_ManualStp36,SP_ManualStp37,SP_ManualStp38,SP_ManualStp39,
	SP_ManualStp40:=2040,SP_ManualStp41,SP_ManualStp42,SP_ManualStp43,SP_ManualStp44,SP_ManualStp45,SP_ManualStp46,SP_ManualStp47,SP_ManualStp48,SP_ManualStp49,
	SP_ManualStp50:=2050,SP_ManualStp51,SP_ManualStp52,SP_ManualStp53,SP_ManualStp54,SP_ManualStp55,SP_ManualStp56,SP_ManualStp57,SP_ManualStp58,SP_ManualStp59,
	SP_ManualStp60:=2060,SP_ManualStp61,SP_ManualStp62,SP_ManualStp63,SP_ManualStp64,SP_ManualStp65,SP_ManualStp66,SP_ManualStp67,SP_ManualStp68,SP_ManualStp69,
	SP_ManualStp70:=2070,SP_ManualStp71,SP_ManualStp72,SP_ManualStp73,SP_ManualStp74,SP_ManualStp75,SP_ManualStp76,SP_ManualStp77,SP_ManualStp78,SP_ManualStp79,
	SP_ManualStp80:=2080,SP_ManualStp81,SP_ManualStp82,SP_ManualStp83,SP_ManualStp84,SP_ManualStp85,SP_ManualStp86,SP_ManualStp87,SP_ManualStp88,SP_ManualStp89,
	SP_ManualStp90:=2090,SP_ManualStp91,SP_ManualStp92,SP_ManualStp93,SP_ManualStp94,SP_ManualStp95,SP_ManualStp96,SP_ManualStp97,SP_ManualStp98,SP_ManualStp99
);
END_TYPE

// ---- Data types/TOperatorReq.TcDUT
{attribute 'pack_mode' := '1'}
TYPE TOperatorReq :
STRUCT
	abFreeLoaderLift			: ARRAY[0..1] OF BOOL;
	bSampleRequest			: BOOL;
END_STRUCT
END_TYPE

// ---- Data types/TPartData.TcDUT
{attribute 'pack_mode' := '1'}
TYPE TPartData :
STRUCT
	bPartPresent			: BOOL;
	ePartSide			: TPearlingSide;
	bToReject			: BOOL;
	bSample				: BOOL;
	abHasPearls			: ARRAY[0..1,0..1] OF BOOL;			(* 1st index is left or right spindle, 2nd is top/bottom *)
	abPearlingDone		: ARRAY[0..1,0..1] OF BOOL;
	anLastPearlIndexDone	: ARRAY[0..1,0..1] OF UINT;
	abBadPearling		: ARRAY[0..1,0..1] OF BOOL;
	dwPlateInQRCode		: DWORD;
	iPlateInPos			: INT;
	dwPlateOutQRCode	: DWORD;
	iPlateOutPos			: INT;
	dwProductionTime	: DWORD;
	dwProductionInTime	: DWORD;
	dwProductionOutTime	: DWORD;
END_STRUCT
END_TYPE

// ---- Data types/TPartDataMMI.TcDUT
{attribute 'pack_mode' := '1'}
TYPE TPartDataMMI :
STRUCT
	lrPartOffsetZLiftTake				: LREAL;
	lrPartOffsetZLiftBadTake			: LREAL;
	lrPartOffsetZLiftDrop				: LREAL;
	lrPartOffsetThetaLiftDrop			: LREAL;
	lrPartOffsetXLiftDrop			: LREAL;
	lrPartOffsetYLiftDrop			: LREAL;
	lrPartOffsetZLayeringTake			: LREAL;
	lrPartOffsetZLayeringDrop			: LREAL;
	lrPartOffsetZTurnOverDrop			: LREAL;
	lrPartOffsetZCleaning				: LREAL;
	alrSensorZOffset					: ARRAY[0..1] OF TPositionXY;
	alrPartOffsetLayering				: ARRAY[0..1] OF TPositionXY;
	lrPartAndLayeringHeight			: LREAL;
	lrPartAndHeadHeight				: LREAL;
	lrLayeringAndPartAndHeadHeight	: LREAL;
	lrHeadSusPartHeadSousHeight		: LREAL;
	lrPlateZOffsetForLift				: LREAL;
	THeadOffset						: TPositionXY;
	eDropModeTable					: TLoaderDropMode;
	eDropModeTurnOver				: TLoaderDropMode;
	eTakeModeLift					: TLoaderTakeMode;
	bDropInBox						: BOOL;
END_STRUCT
END_TYPE

// ---- Data types/TPearlingAxis.TcDUT
TYPE TPearlingAxis :
	(
		PA_X := 0,
		PA_Y,
		PA_Z1,
		PA_Z2
	);
END_TYPE

// ---- Data types/TPearlingData.TcDUT
{attribute 'pack_mode' := '1'}
TYPE TPearlingData :
STRUCT
		THead 	: ARRAY[PH_Left..PH_Right] OF TPearlingDataHead;
END_STRUCT
END_TYPE

// ---- Data types/TPearlingDataHead.TcDUT
{attribute 'pack_mode' := '1'}
TYPE TPearlingDataHead :
STRUCT
	aDataPerlage		: ARRAY[0..C_MAX_NB_OF_PEARLS] OF TPearlsTable;
	nNbOfPearls			: UINT;
	lrSecurityZ			: LREAL;
	iDispersionXY		: INT;
	iWeight				: INT;
	iDispersionZ			: INT;
	iSharpenFreq			: INT;
	iMCRSpeed			: INT;
	iPearlingTime		: INT;
END_STRUCT
END_TYPE

// ---- Data types/TPearlingDebug.TcDUT
{attribute 'pack_mode' := '1'}
TYPE TPearlingDebug :
	STRUCT
		iStep				: INT;
		iStickStep			: INT;
		aiProbingStep		: ARRAY[0..1] OF INT;
		abOpenChuck		: ARRAY[0..1] OF BOOL;
		abChangeStick		: ARRAY[0..1] OF BOOL;
		abSharpenStick		: ARRAY[0..1] OF BOOL;
		abUseSpindle		: ARRAY[0..1] OF BOOL;
	END_STRUCT
END_TYPE

// ---- Data types/TPearlingHead.TcDUT
TYPE TPearlingHead :
	(
		PH_Left := 0,
		PH_Right
	);
END_TYPE

// ---- Data types/TPearlingSide.TcDUT
TYPE TPearlingSide :
	(
		PS_SUS := 0,
		PS_SOUS
	);
END_TYPE

// ---- Data types/TPearlingTeachPos.TcDUT
TYPE TPearlingTeachPos :
	(
		PTP_TableSideAPosZ1 := 0,
		PTP_TableSideAPosZ2,
		PTP_TableSideBPosZ1,
		PTP_TableSideBPosZ2,
		PTP_BarrelPosZ1,
		PTP_BarrelPosZ2,
		PTP_RejectPosZ1,
		PTP_RejectPosZ2,
		PTP_Sharpen,
		PTP_WeightCalibrationPosZ1,
		PTP_WeightCalibrationPosZ2,
		PTP_END
	);
END_TYPE

// ---- Data types/TPearlsArea.TcDUT
{attribute 'pack_mode' := '1'}
TYPE TPearlsArea :
STRUCT
	iNbOfPearls		: INT;
	iFirstPearl		: INT;
END_STRUCT
END_TYPE

// ---- Data types/TPearlsTable.TcDUT
{attribute 'pack_mode' := '1'}
TYPE TPearlsTable :
STRUCT
	iArea			: INT;
	bXYDispersion	: BOOL;
	bForceSharpen	: BOOL;
	bDisable			: BOOL;
	bMoveToSafe	: BOOL;
	lrX				: LREAL;
	lrY				: LREAL;
	lrZ				: LREAL;
	lrRate			: LREAL;
END_STRUCT
END_TYPE

